C01821=1123.356,380.841,-87.477,-176.868,11.252,149.471
C01822=1123.352,381.088,-87.514,-176.865,11.254,149.471
C01823=1123.349,381.335,-87.552,-176.862,11.256,149.470
C01824=1123.345,381.582,-87.589,-176.859,11.259,149.470
C01825=1123.342,381.830,-87.627,-176.856,11.262,149.470
C01826=1123.338,382.077,-87.664,-176.854,11.263,149.470
C01827=1123.334,382.325,-87.702,-176.851,11.266,149.470
C01828=1123.330,382.571,-87.740,-176.848,11.269,149.470
C01829=1123.326,382.818,-87.777,-176.845,11.272,149.470
C01830=1123.323,383.066,-87.814,-176.842,11.274,149.470
C01831=1123.319,383.313,-87.851,-176.839,11.276,149.470
C01832=1123.315,383.560,-87.889,-176.837,11.278,149.470
C01833=1123.312,383.807,-87.927,-176.835,11.280,149.470
C01834=1123.308,384.054,-87.964,-176.833,11.283,149.470
C01835=1123.304,384.301,-88.002,-176.832,11.284,149.470
C01836=1123.301,384.548,-88.040,-176.830,11.286,149.470
C01837=1123.296,384.796,-88.077,-176.828,11.289,149.470
C01838=1123.293,385.042,-88.115,-176.826,11.291,149.470
C01839=1123.289,385.290,-88.153,-176.824,11.292,149.470
C01840=1123.286,385.536,-88.190,-176.822,11.295,149.470
C01841=1123.282,385.784,-88.227,-176.820,11.297,149.470
C01842=1123.278,386.031,-88.265,-176.819,11.299,149.471
C01843=1123.274,386.278,-88.303,-176.817,11.301,149.471
C01844=1123.271,386.525,-88.341,-176.815,11.303,149.471
C01845=1123.267,386.773,-88.378,-176.814,11.306,149.471
C01846=1123.263,387.019,-88.416,-176.812,11.308,149.471
C01847=1123.260,387.267,-88.454,-176.810,11.310,149.471
C01848=1123.256,387.513,-88.492,-176.809,11.312,149.471
C01849=1123.252,387.761,-88.530,-176.807,11.314,149.471
C01850=1123.248,388.008,-88.567,-176.805,11.317,149.472
C01851=1123.245,388.255,-88.605,-176.803,11.319,149.472
C01852=1123.241,388.502,-88.642,-176.802,11.321,149.472
C01853=1123.238,388.714,-88.675,-176.800,11.323,149.472
C01854=1123.234,388.926,-88.707,-176.799,11.325,149.472
C01855=1123.232,389.138,-88.740,-176.797,11.328,149.473
C01856=1123.228,389.350,-88.773,-176.796,11.329,149.473
C01857=1123.226,389.562,-88.805,-176.795,11.332,149.473
C01858=1123.222,389.775,-88.837,-176.793,11.333,149.473
C01859=1123.219,389.987,-88.870,-176.792,11.336,149.473
C01860=1123.216,390.199,-88.902,-176.791,11.338,149.473
C01861=1123.212,390.446,-88.940,-176.789,11.340,149.474
C01862=1123.209,390.694,-88.978,-176.788,11.343,149.474
C01863=1123.205,390.940,-89.016,-176.786,11.345,149.474
C01864=1123.202,391.188,-89.054,-176.784,11.348,149.475
C01865=1123.197,391.434,-89.092,-176.783,11.351,149.475
C01866=1123.194,391.682,-89.130,-176.781,11.354,149.475
C01867=1123.190,391.928,-89.168,-176.780,11.356,149.475
C01868=1123.187,392.176,-89.206,-176.779,11.358,149.476
C01869=1123.183,392.423,-89.244,-176.778,11.361,149.476
C01870=1123.180,392.670,-89.282,-176.776,11.363,149.476
C01871=1123.176,392.917,-89.320,-176.775,11.366,149.477
C01872=1123.172,393.164,-89.358,-176.773,11.369,149.477
C01873=1123.169,393.411,-89.396,-176.772,11.372,149.477
C01874=1123.164,393.658,-89.434,-176.770,11.374,149.478
C01875=1123.161,393.905,-89.472,-176.769,11.377,149.478
C01876=1123.158,394.153,-89.510,-176.768,11.380,149.479
C01877=1123.153,394.399,-89.548,-176.766,11.383,149.479
C01878=1123.150,394.647,-89.586,-176.765,11.386,149.479
C01879=1123.146,394.893,-89.623,-176.764,11.388,149.480
C01880=1123.142,395.141,-89.662,-176.762,11.392,149.480
C01881=1123.139,395.388,-89.701,-176.761,11.395,149.481
C01882=1123.135,395.634,-89.739,-176.759,11.398,149.481
C01883=1123.132,395.882,-89.777,-176.758,11.401,149.482
C01884=1123.128,396.128,-89.814,-176.757,11.404,149.482
C01885=1123.124,396.376,-89.853,-176.756,11.407,149.482
C01886=1123.121,396.623,-89.891,-176.755,11.410,149.483
C01887=1123.116,396.870,-89.929,-176.753,11.413,149.483
C01888=1123.113,397.117,-89.967,-176.752,11.416,149.484
C01889=1123.110,397.364,-90.005,-176.751,11.419,149.484
C01890=1123.106,397.611,-90.044,-176.750,11.422,149.485
C01891=1123.103,397.858,-90.082,-176.748,11.425,149.485
C01892=1123.099,398.106,-90.120,-176.748,11.429,149.486
C01893=1123.095,398.352,-90.158,-176.747,11.432,149.487
C01894=1123.091,398.599,-90.197,-176.746,11.435,149.487
C01895=1123.088,398.846,-90.235,-176.744,11.439,149.488
C01896=1123.083,399.093,-90.273,-176.743,11.442,149.488
C01897=1123.080,399.341,-90.311,-176.742,11.445,149.489
C01898=1123.077,399.587,-90.350,-176.741,11.448,149.490
C01899=1123.073,399.834,-90.388,-176.740,11.452,149.490
C01900=1123.070,400.081,-90.426,-176.739,11.455,149.491
C01901=1123.066,400.328,-90.465,-176.738,11.459,149.492
C01902=1123.062,400.575,-90.503,-176.737,11.462,149.492
C01903=1123.058,400.823,-90.541,-176.736,11.466,149.493
C01904=1123.055,401.070,-90.579,-176.735,11.469,149.493
C01905=1123.051,401.316,-90.618,-176.734,11.473,149.494
C01906=1123.048,401.563,-90.656,-176.733,11.477,149.495
C01907=1123.044,401.811,-90.694,-176.732,11.480,149.496
C01908=1123.040,402.057,-90.733,-176.732,11.483,149.496
C01909=1123.037,402.270,-90.766,-176.731,11.486,149.497
C01910=1123.034,402.482,-90.799,-176.730,11.490,149.498
C01911=1123.031,402.693,-90.832,-176.729,11.493,149.498
C01912=1123.028,402.906,-90.865,-176.729,11.496,149.499
C01913=1123.024,403.117,-90.898,-176.728,11.500,149.500
C01914=1123.021,403.330,-90.931,-176.727,11.503,149.500
C01915=1123.018,403.541,-90.964,-176.726,11.506,149.501
C01916=1123.015,403.753,-90.997,-176.725,11.509,149.501
C01917=1123.011,404.000,-91.035,-176.725,11.513,149.502
C01918=1123.008,404.247,-91.075,-176.724,11.517,149.503
C01919=1123.005,404.495,-91.112,-176.723,11.521,149.504
C01920=1123.000,404.741,-91.151,-176.722,11.525,149.505
C01921=1122.997,404.988,-91.189,-176.722,11.529,149.506
C01922=1122.993,405.236,-91.228,-176.721,11.533,149.507
C01923=1122.990,405.482,-91.266,-176.720,11.537,149.507
C01924=1122.986,405.729,-91.305,-176.719,11.541,149.508
C01925=1122.982,405.976,-91.344,-176.719,11.545,149.509
C01926=1122.979,406.224,-91.382,-176.719,11.550,149.510
C01927=1122.976,406.470,-91.421,-176.718,11.553,149.511
C01928=1122.972,406.716,-91.459,-176.717,11.558,149.512
C01929=1122.968,406.964,-91.498,-176.716,11.562,149.513
C01930=1122.964,407.211,-91.537,-176.716,11.566,149.514
C01931=1122.961,407.458,-91.575,-176.716,11.571,149.515
C01932=1122.958,407.705,-91.614,-176.715,11.574,149.516
C01933=1122.953,407.952,-91.653,-176.715,11.579,149.517
C01934=1122.950,408.199,-91.691,-176.714,11.584,149.518
C01935=1122.947,408.446,-91.730,-176.714,11.587,149.519
C01936=1122.943,408.693,-91.769,-176.713,11.592,149.520
C01937=1122.940,408.940,-91.808,-176.713,11.597,149.521
C01938=1122.935,409.187,-91.846,-176.712,11.602,149.522
C01939=1122.932,409.434,-91.885,-176.712,11.606,149.523
C01940=1122.929,409.680,-91.924,-176.712,11.611,149.524
C01941=1122.925,409.928,-91.962,-176.711,11.615,149.526
C01942=1122.921,410.175,-92.001,-176.710,11.620,149.527
C01943=1122.918,410.421,-92.040,-176.711,11.624,149.528
C01944=1122.914,410.669,-92.078,-176.710,11.629,149.529
C01945=1122.910,410.915,-92.118,-176.710,11.634,149.530
C01946=1122.907,411.162,-92.157,-176.709,11.639,149.531
C01947=1122.903,411.410,-92.195,-176.709,11.644,149.532
C01948=1122.900,411.657,-92.234,-176.709,11.649,149.534
C01949=1122.896,411.903,-92.273,-176.708,11.654,149.535
C01950=1122.892,412.150,-92.312,-176.709,11.658,149.536
C01951=1122.889,412.397,-92.350,-176.708,11.663,149.537
C01952=1122.885,412.644,-92.389,-176.708,11.668,149.538
C01953=1122.882,412.891,-92.429,-176.708,11.673,149.540
C01954=1122.878,413.138,-92.468,-176.708,11.678,149.541
C01955=1122.875,413.385,-92.506,-176.707,11.683,149.542
C01956=1122.871,413.632,-92.545,-176.707,11.688,149.544
C01957=1122.867,413.879,-92.584,-176.707,11.693,149.545
C01958=1122.865,414.126,-92.623,-176.707,11.699,149.546
C01959=1122.862,414.373,-92.662,-176.707,11.704,149.548
C01960=1122.860,414.620,-92.700,-176.707,11.709,149.549
C01961=1122.859,414.866,-92.739,-176.707,11.714,149.550
C01962=1122.858,415.114,-92.778,-176.707,11.720,149.552
C01963=1122.858,415.361,-92.816,-176.707,11.725,149.553
C01964=1122.858,415.608,-92.855,-176.707,11.730,149.555
C01965=1122.859,415.819,-92.887,-176.707,11.735,149.556
C01966=1122.860,416.031,-92.920,-176.708,11.740,149.557
C01967=1122.862,416.243,-92.953,-176.707,11.745,149.558
C01968=1122.864,416.455,-92.986,-176.708,11.749,149.560
C01969=1122.865,416.667,-93.019,-176.708,11.754,149.561
C01970=1122.869,416.878,-93.052,-176.708,11.759,149.562
C01971=1122.872,417.090,-93.084,-176.708,11.764,149.564
C01972=1122.876,417.302,-93.116,-176.709,11.768,149.565
C01973=1122.457,417.301,-93.179,-176.701,11.773,149.564
C01974=1122.453,417.090,-93.147,-176.701,11.768,149.563
C01975=1122.449,416.878,-93.114,-176.701,11.763,149.561
C01976=1122.447,416.667,-93.081,-176.700,11.759,149.560
C01977=1122.445,416.455,-93.049,-176.700,11.753,149.559
C01978=1122.443,416.243,-93.016,-176.700,11.749,149.558
C01979=1122.441,416.031,-92.983,-176.700,11.744,149.556
C01980=1122.440,415.819,-92.950,-176.700,11.740,149.555
C01981=1122.439,415.607,-92.917,-176.700,11.735,149.554
C01982=1122.438,415.360,-92.879,-176.700,11.730,149.553
C01983=1122.439,415.113,-92.840,-176.700,11.724,149.551
C01984=1122.440,414.867,-92.801,-176.700,11.719,149.550
C01985=1122.441,414.620,-92.763,-176.700,11.714,149.548
C01986=1122.443,414.373,-92.724,-176.700,11.709,149.547
C01987=1122.445,414.125,-92.685,-176.700,11.703,149.546
C01988=1122.448,413.879,-92.647,-176.701,11.697,149.544
C01989=1122.452,413.632,-92.607,-176.701,11.692,149.543
C01990=1122.455,413.385,-92.568,-176.701,11.687,149.542
C01991=1122.458,413.138,-92.529,-176.701,11.682,149.540
C01992=1122.462,412.891,-92.490,-176.701,11.677,149.539
C01993=1122.466,412.643,-92.452,-176.702,11.672,149.538
C01994=1122.470,412.397,-92.413,-176.702,11.667,149.537
C01995=1122.473,412.150,-92.374,-176.702,11.662,149.536
C01996=1122.476,411.904,-92.335,-176.703,11.657,149.534
C01997=1122.480,411.656,-92.296,-176.703,11.652,149.533
C01998=1122.484,411.409,-92.257,-176.703,11.647,149.532
C01999=1122.488,411.162,-92.218,-176.703,11.643,149.531
C02000=1122.490,410.915,-92.179,-176.703,11.638,149.529
C02001=1122.495,410.668,-92.141,-176.704,11.633,149.528
C02002=1122.499,410.422,-92.102,-176.704,11.628,149.527
C02003=1122.501,410.175,-92.063,-176.705,11.623,149.526
C02004=1122.505,409.927,-92.025,-176.705,11.618,149.525
C02005=1122.509,409.680,-91.985,-176.706,11.614,149.524
C02006=1122.513,409.433,-91.946,-176.706,11.610,149.523
C02007=1122.516,409.187,-91.909,-176.706,11.605,149.522
C02008=1122.520,408.940,-91.869,-176.707,11.600,149.521
C02009=1122.524,408.693,-91.830,-176.708,11.596,149.520
C02010=1122.527,408.446,-91.792,-176.708,11.591,149.518
C02011=1122.530,408.199,-91.753,-176.708,11.587,149.517
C02012=1122.535,407.952,-91.714,-176.709,11.582,149.517
C02013=1122.538,407.705,-91.676,-176.710,11.578,149.515
C02014=1122.541,407.458,-91.637,-176.710,11.574,149.515
C02015=1122.545,407.211,-91.598,-176.711,11.570,149.514
C02016=1122.548,406.964,-91.560,-176.712,11.565,149.512
C02017=1122.552,406.718,-91.521,-176.713,11.560,149.512
C02018=1122.556,406.470,-91.482,-176.713,11.557,149.511
C02019=1122.559,406.223,-91.444,-176.714,11.552,149.510
C02020=1122.563,405.976,-91.405,-176.714,11.549,149.509
C02021=1122.567,405.730,-91.367,-176.715,11.544,149.508
C02022=1122.571,405.482,-91.328,-176.716,11.540,149.507
C02023=1122.574,405.235,-91.289,-176.716,11.536,149.506
C02024=1122.577,404.988,-91.251,-176.717,11.532,149.505
C02025=1122.581,404.741,-91.212,-176.718,11.528,149.504
C02026=1122.585,404.495,-91.174,-176.719,11.524,149.504
C02027=1122.588,404.248,-91.135,-176.719,11.520,149.503
C02028=1122.592,404.000,-91.096,-176.720,11.516,149.502
C02029=1122.595,403.753,-91.058,-176.721,11.512,149.501
C02030=1122.599,403.541,-91.025,-176.722,11.509,149.500
C02031=1122.602,403.329,-90.992,-176.722,11.506,149.500
C02032=1122.605,403.118,-90.958,-176.723,11.502,149.499
C02033=1122.609,402.905,-90.926,-176.724,11.499,149.498
C02034=1122.611,402.694,-90.893,-176.725,11.496,149.498
C02035=1122.614,402.482,-90.861,-176.726,11.493,149.497
C02036=1122.618,402.270,-90.827,-176.726,11.489,149.496
C02037=1122.621,402.058,-90.794,-176.727,11.486,149.496
C02038=1122.625,401.810,-90.755,-176.729,11.482,149.495
C02039=1122.628,401.563,-90.718,-176.729,11.479,149.495
C02040=1122.632,401.316,-90.678,-176.730,11.475,149.494
C02041=1122.635,401.070,-90.641,-176.731,11.471,149.493
C02042=1122.639,400.823,-90.601,-176.732,11.468,149.492
C02043=1122.642,400.575,-90.564,-176.733,11.464,149.492
C02044=1122.647,400.329,-90.525,-176.735,11.461,149.491
C02045=1122.650,400.081,-90.487,-176.735,11.458,149.490
C02046=1122.653,399.834,-90.448,-176.736,11.454,149.490
C02047=1122.657,399.588,-90.411,-176.738,11.450,149.489
C02048=1122.661,399.340,-90.372,-176.738,11.447,149.489
C02049=1122.664,399.094,-90.333,-176.739,11.444,149.488
C02050=1122.669,398.847,-90.295,-176.741,11.440,149.487
C02051=1122.672,398.599,-90.257,-176.742,11.437,149.487
C02052=1122.675,398.352,-90.219,-176.743,11.434,149.486
C02053=1122.679,398.106,-90.180,-176.744,11.431,149.486
C02054=1122.682,397.859,-90.143,-176.746,11.427,149.485
C02055=1122.686,397.611,-90.104,-176.747,11.424,149.485
C02056=1122.690,397.364,-90.066,-176.748,11.421,149.484
C02057=1122.694,397.117,-90.028,-176.749,11.418,149.484
C02058=1122.697,396.870,-89.989,-176.750,11.415,149.483
C02059=1122.701,396.623,-89.951,-176.752,11.411,149.483
C02060=1122.705,396.376,-89.913,-176.753,11.408,149.482
C02061=1122.708,396.129,-89.876,-176.754,11.405,149.482
C02062=1122.712,395.882,-89.837,-176.756,11.403,149.481
C02063=1122.715,395.635,-89.799,-176.757,11.400,149.481
C02064=1122.720,395.388,-89.761,-176.758,11.397,149.480
C02065=1122.723,395.141,-89.722,-176.759,11.394,149.480
C02066=1122.726,394.894,-89.684,-176.761,11.390,149.479
C02067=1122.731,394.647,-89.646,-176.762,11.387,149.479
C02068=1122.734,394.400,-89.608,-176.763,11.384,149.479
C02069=1122.738,394.153,-89.571,-176.765,11.382,149.478
C02070=1122.742,393.906,-89.532,-176.766,11.379,149.478
C02071=1122.745,393.658,-89.494,-176.768,11.376,149.477
C02072=1122.749,393.411,-89.456,-176.769,11.373,149.477
C02073=1122.752,393.164,-89.418,-176.771,11.371,149.477
C02074=1122.756,392.918,-89.380,-176.772,11.368,149.476
C02075=1122.760,392.670,-89.342,-176.773,11.365,149.476
C02076=1122.764,392.423,-89.304,-176.775,11.363,149.476
C02077=1122.767,392.176,-89.266,-176.776,11.360,149.476
C02078=1122.771,391.929,-89.228,-176.778,11.357,149.475
C02079=1122.775,391.682,-89.190,-176.779,11.354,149.475
C02080=1122.778,391.435,-89.152,-176.781,11.352,149.475
C02081=1122.782,391.188,-89.115,-176.782,11.349,149.474
C02082=1122.786,390.941,-89.076,-176.784,11.347,149.474
C02083=1122.790,390.694,-89.039,-176.786,11.344,149.474
C02084=1122.793,390.447,-89.001,-176.787,11.341,149.473
C02085=1122.796,390.199,-88.963,-176.789,11.339,149.473
C02086=1122.799,389.987,-88.930,-176.790,11.337,149.473
C02087=1122.803,389.775,-88.898,-176.792,11.335,149.473
C02088=1122.806,389.563,-88.866,-176.793,11.333,149.473
C02089=1122.809,389.351,-88.832,-176.795,11.330,149.473
C02090=1122.812,389.139,-88.800,-176.796,11.329,149.472
C02091=1122.815,388.927,-88.768,-176.797,11.326,149.472
C02092=1122.819,388.715,-88.736,-176.799,11.325,149.472
C02093=1122.822,388.503,-88.704,-176.800,11.322,149.472
C02094=1122.826,388.255,-88.665,-176.801,11.320,149.472
C02095=1122.829,388.008,-88.627,-176.803,11.318,149.471
C02096=1122.833,387.762,-88.590,-176.805,11.316,149.471
C02097=1122.836,387.514,-88.552,-176.807,11.313,149.471
C02098=1122.840,387.267,-88.515,-176.809,11.311,149.471
C02099=1122.844,387.019,-88.476,-176.811,11.309,149.471
C02100=1122.848,386.773,-88.439,-176.812,11.307,149.471
C02101=1122.851,386.526,-88.401,-176.814,11.305,149.471
C02102=1122.855,386.278,-88.364,-176.816,11.302,149.471
C02103=1122.858,386.031,-88.326,-176.817,11.300,149.470
C02104=1122.863,385.784,-88.288,-176.819,11.298,149.470
C02105=1122.866,385.537,-88.250,-176.821,11.296,149.470
C02106=1122.870,385.290,-88.213,-176.822,11.294,149.470
C02107=1122.874,385.043,-88.175,-176.825,11.292,149.470
C02108=1122.877,384.796,-88.137,-176.827,11.289,149.470
C02109=1122.881,384.549,-88.100,-176.829,11.287,149.470
C02110=1122.884,384.302,-88.063,-176.830,11.286,149.470
C02111=1122.889,384.055,-88.024,-176.832,11.283,149.470
C02112=1122.892,383.807,-87.986,-176.834,11.281,149.470
C02113=1122.896,383.560,-87.950,-176.836,11.279,149.470
C02114=1122.899,383.313,-87.912,-176.838,11.277,149.470
C02115=1122.903,383.066,-87.874,-176.841,11.275,149.470
C02116=1122.906,382.818,-87.837,-176.844,11.272,149.470
C02117=1122.910,382.572,-87.799,-176.847,11.270,149.470
C02118=1122.914,382.325,-87.762,-176.850,11.267,149.470
C02119=1122.918,382.077,-87.725,-176.852,11.265,149.470
C02120=1122.921,381.831,-87.687,-176.855,11.262,149.470
C02121=1122.926,381.583,-87.649,-176.858,11.259,149.470
C02122=1122.929,381.336,-87.612,-176.862,11.257,149.471
C02123=1122.933,381.088,-87.574,-176.864,11.255,149.471
C02124=1122.937,380.842,-87.537,-176.867,11.252,149.471
C02125=1122.941,380.594,-87.500,-176.870,11.250,149.471
C02126=1122.944,380.347,-87.462,-176.873,11.247,149.471
C02127=1122.948,380.100,-87.425,-176.876,11.244,149.471
C02128=1122.952,379.853,-87.388,-176.879,11.243,149.471
C02129=1122.955,379.606,-87.350,-176.882,11.240,149.471
C02130=1122.959,379.359,-87.313,-176.885,11.237,149.471
C02131=1122.963,379.111,-87.275,-176.888,11.234,149.471
C02132=1122.966,378.865,-87.238,-176.891,11.233,149.472
C02133=1122.970,378.617,-87.201,-176.894,11.230,149.472
C02134=1122.974,378.369,-87.164,-176.897,11.227,149.472
C02135=1122.978,378.123,-87.126,-176.900,11.225,149.472
C02136=1122.982,377.876,-87.089,-176.902,11.223,149.472
C02137=1122.985,377.628,-87.053,-176.906,11.220,149.472
C02138=1122.988,377.382,-87.015,-176.909,11.218,149.473
C02139=1122.992,377.134,-86.978,-176.912,11.215,149.473
C02140=1122.996,376.886,-86.941,-176.915,11.213,149.473
C02141=1123.000,376.640,-86.904,-176.918,11.211,149.473
C02142=1123.004,376.427,-86.872,-176.921,11.208,149.473
C02143=1123.007,376.216,-86.840,-176.923,11.206,149.473
C02144=1123.010,376.003,-86.809,-176.926,11.204,149.473
C02145=1123.013,375.791,-86.776,-176.928,11.203,149.474
C02146=1123.016,375.579,-86.744,-176.931,11.200,149.474
C02147=1123.019,375.366,-86.713,-176.934,11.198,149.474
C02148=1123.023,375.155,-86.681,-176.936,11.196,149.474
C02149=1123.026,374.942,-86.649,-176.939,11.195,149.474
C02150=1123.030,374.694,-86.612,-176.942,11.192,149.474
C02151=1123.033,374.447,-86.575,-176.945,11.190,149.475
C02152=1123.037,374.200,-86.538,-176.948,11.187,149.475
C02153=1123.041,373.953,-86.502,-176.952,11.184,149.475
C02154=1123.045,373.705,-86.464,-176.954,11.183,149.475
C02155=1123.049,373.458,-86.427,-176.958,11.180,149.475
C02156=1123.052,373.211,-86.391,-176.961,11.178,149.475
C02157=1123.056,372.964,-86.354,-176.964,11.175,149.476
C02158=1123.060,372.716,-86.317,-176.968,11.173,149.476
C02159=1123.064,372.469,-86.280,-176.970,11.171,149.476
C02160=1123.067,372.222,-86.244,-176.974,11.169,149.476
C02161=1123.071,371.975,-86.206,-176.977,11.166,149.477
C02162=1123.075,371.728,-86.170,-176.980,11.163,149.477
C02163=1123.078,371.480,-86.132,-176.983,11.161,149.477
C02164=1123.082,371.233,-86.097,-176.986,11.158,149.477
C02165=1123.086,370.986,-86.060,-176.989,11.157,149.477
C02166=1123.090,370.738,-86.023,-176.992,11.154,149.477
C02167=1123.094,370.492,-85.987,-176.996,11.152,149.478
C02168=1123.097,370.244,-85.950,-176.999,11.149,149.478
C02169=1123.101,369.996,-85.913,-177.002,11.147,149.478
C02170=1123.105,369.750,-85.876,-177.005,11.144,149.478
C02171=1123.109,369.502,-85.840,-177.009,11.143,149.479
C02172=1123.113,369.255,-85.803,-177.012,11.140,149.479
C02173=1123.116,369.008,-85.766,-177.015,11.138,149.479
C02174=1123.120,368.760,-85.729,-177.018,11.135,149.479
C02175=1123.124,368.513,-85.693,-177.022,11.133,149.479
C02176=1123.127,368.266,-85.657,-177.025,11.130,149.480
C02177=1123.131,368.019,-85.620,-177.028,11.128,149.480
C02178=1123.135,367.772,-85.584,-177.032,11.125,149.480
C02179=1123.139,367.524,-85.548,-177.034,11.124,149.480
C02180=1123.143,367.277,-85.511,-177.038,11.121,149.481
C02181=1123.147,367.030,-85.474,-177.041,11.119,149.481
C02182=1123.150,366.782,-85.437,-177.044,11.116,149.481
C02183=1123.154,366.534,-85.402,-177.048,11.114,149.481
C02184=1123.158,366.287,-85.365,-177.051,11.112,149.482
C02185=1123.161,366.040,-85.329,-177.055,11.109,149.482
C02186=1123.166,365.793,-85.292,-177.058,11.107,149.482
C02187=1123.169,365.546,-85.256,-177.061,11.104,149.482
C02188=1123.173,365.298,-85.219,-177.064,11.103,149.483
C02189=1123.177,365.051,-85.184,-177.067,11.100,149.483
C02190=1123.181,364.804,-85.147,-177.071,11.098,149.483
C02191=1123.185,364.556,-85.111,-177.074,11.096,149.483
C02192=1123.189,364.309,-85.074,-177.077,11.093,149.484
C02193=1123.192,364.062,-85.038,-177.081,11.091,149.484
C02194=1123.196,363.814,-85.002,-177.084,11.088,149.484
C02195=1123.199,363.567,-84.965,-177.088,11.086,149.484
C02196=1123.204,363.319,-84.929,-177.091,11.084,149.485
C02197=1123.207,363.072,-84.893,-177.094,11.081,149.485
C02198=1123.211,362.826,-84.857,-177.098,11.079,149.485
C02199=1123.215,362.580,-84.821,-177.101,11.076,149.485
C02200=1123.218,362.332,-84.786,-177.105,11.074,149.486
C02201=1123.222,362.086,-84.750,-177.108,11.071,149.486
C02202=1123.226,361.839,-84.714,-177.111,11.069,149.486
C02203=1123.230,361.593,-84.678,-177.115,11.067,149.486
C02204=1123.234,361.347,-84.642,-177.118,11.064,149.486
C02205=1123.237,361.100,-84.605,-177.122,11.062,149.487
C02206=1123.241,360.852,-84.569,-177.125,11.059,149.487
C02207=1123.245,360.605,-84.534,-177.128,11.057,149.487
C02208=1123.248,360.358,-84.498,-177.131,11.055,149.488
C02209=1123.253,360.110,-84.461,-177.135,11.052,149.488
C02210=1123.257,359.863,-84.426,-177.138,11.050,149.488
C02211=1123.260,359.616,-84.390,-177.142,11.047,149.488
C02212=1123.264,359.368,-84.354,-177.145,11.045,149.489
C02213=1123.268,359.120,-84.318,-177.148,11.043,149.489
C02214=1123.272,358.874,-84.283,-177.152,11.040,149.489
C02215=1123.276,358.627,-84.246,-177.155,11.038,149.489
C02216=1123.279,358.379,-84.211,-177.159,11.035,149.490
C02217=1123.284,358.131,-84.175,-177.162,11.033,149.490
C02218=1123.287,357.884,-84.139,-177.166,11.031,149.490
C02219=1123.291,357.636,-84.104,-177.169,11.028,149.490
C02220=1123.294,357.389,-84.067,-177.172,11.026,149.491
C02221=1123.299,357.142,-84.031,-177.176,11.023,149.491
C02222=1123.302,356.928,-84.001,-177.179,11.021,149.491
C02223=1123.305,356.715,-83.970,-177.182,11.019,149.491
C02224=1123.309,356.502,-83.940,-177.185,11.017,149.492
C02225=1123.312,356.289,-83.909,-177.188,11.015,149.492
C02226=1123.315,356.076,-83.878,-177.191,11.013,149.492
C02227=1123.319,355.863,-83.847,-177.194,11.010,149.492
C02228=1123.322,355.649,-83.817,-177.197,11.009,149.493
C02229=1123.325,355.435,-83.786,-177.200,11.006,149.493
C02230=1123.329,355.189,-83.750,-177.204,11.004,149.493
C02231=1123.333,354.941,-83.715,-177.207,11.001,149.493
C02232=1123.336,354.694,-83.679,-177.210,10.999,149.493
C02233=1123.341,354.446,-83.643,-177.214,10.997,149.494
C02234=1123.344,354.198,-83.608,-177.217,10.994,149.494
C02235=1123.348,353.951,-83.572,-177.221,10.991,149.494
C02236=1123.352,353.704,-83.537,-177.224,10.988,149.495
C02237=1123.356,353.456,-83.501,-177.228,10.986,149.495
C02238=1123.360,353.209,-83.466,-177.231,10.984,149.495
C02239=1123.363,352.961,-83.430,-177.235,10.981,149.495
C02240=1123.367,352.713,-83.395,-177.238,10.979,149.496
C02241=1123.371,352.467,-83.360,-177.242,10.976,149.496
C02242=1123.375,352.219,-83.325,-177.246,10.973,149.496
C02243=1123.379,351.972,-83.289,-177.249,10.971,149.496
C02244=1123.382,351.724,-83.254,-177.252,10.969,149.497
C02245=1123.387,351.477,-83.219,-177.256,10.965,149.497
C02246=1123.391,351.229,-83.184,-177.260,10.963,149.497
C02247=1123.394,350.982,-83.148,-177.263,10.960,149.497
C02248=1123.398,350.734,-83.113,-177.267,10.958,149.498
C02249=1123.403,350.487,-83.078,-177.271,10.955,149.498
C02250=1123.406,350.239,-83.043,-177.274,10.953,149.498
C02251=1123.410,349.992,-83.007,-177.277,10.950,149.498
C02252=1123.414,349.745,-82.972,-177.280,10.948,149.499
C02253=1123.418,349.497,-82.937,-177.284,10.944,149.499
C02254=1123.421,349.284,-82.907,-177.287,10.943,149.499
C02255=1123.424,349.072,-82.876,-177.289,10.941,149.499
C02256=1123.428,348.860,-82.847,-177.293,10.938,149.499
C02257=1123.431,348.646,-82.816,-177.295,10.937,149.500
C02258=1123.434,348.434,-82.786,-177.298,10.934,149.500
C02259=1123.438,348.221,-82.756,-177.301,10.932,149.500
C02260=1123.441,348.009,-82.726,-177.304,10.930,149.500
C02261=1123.445,347.796,-82.696,-177.307,10.928,149.500
C02262=1123.448,347.548,-82.660,-177.310,10.925,149.500
C02263=1123.453,347.301,-82.626,-177.313,10.923,149.501
C02264=1123.457,347.054,-82.590,-177.317,10.920,149.501
C02265=1123.460,346.806,-82.556,-177.320,10.918,149.501
C02266=1123.464,346.559,-82.521,-177.323,10.915,149.501
C02267=1123.468,346.311,-82.486,-177.325,10.913,149.501
C02268=1123.472,346.064,-82.451,-177.329,10.911,149.502
C02269=1123.476,345.816,-82.416,-177.332,10.908,149.502
C02270=1123.479,345.569,-82.381,-177.335,10.906,149.502
C02271=1123.484,345.321,-82.347,-177.339,10.903,149.502
C02272=1123.487,345.074,-82.311,-177.342,10.901,149.502
C02273=1123.492,344.826,-82.277,-177.345,10.898,149.503
C02274=1123.496,344.578,-82.242,-177.348,10.896,149.503
C02275=1123.499,344.331,-82.207,-177.352,10.893,149.503
C02276=1123.503,344.084,-82.172,-177.355,10.891,149.503
C02277=1123.507,343.836,-82.138,-177.358,10.888,149.504
C02278=1123.512,343.589,-82.102,-177.361,10.886,149.504
C02279=1123.515,343.341,-82.068,-177.364,10.883,149.504
C02280=1123.519,343.093,-82.033,-177.368,10.881,149.504
C02281=1123.523,342.845,-81.999,-177.371,10.878,149.504
C02282=1123.526,342.598,-81.964,-177.374,10.876,149.505
C02283=1123.531,342.351,-81.930,-177.378,10.873,149.505
C02284=1123.535,342.103,-81.895,-177.380,10.871,149.505
C02285=1123.539,341.856,-81.861,-177.383,10.869,149.505
C02286=1123.542,341.608,-81.825,-177.387,10.866,149.505
C02287=1123.547,341.361,-81.791,-177.390,10.864,149.506
C02288=1123.550,341.113,-81.757,-177.393,10.862,149.506
C02289=1123.555,340.865,-81.722,-177.396,10.859,149.506
C02290=1123.559,340.617,-81.687,-177.399,10.856,149.506
C02291=1123.563,340.370,-81.653,-177.403,10.854,149.506
C02292=1123.567,340.122,-81.619,-177.406,10.851,149.507
C02293=1123.570,339.876,-81.584,-177.409,10.849,149.507
C02294=1123.574,339.627,-81.549,-177.412,10.846,149.507
C02295=1123.579,339.380,-81.515,-177.416,10.844,149.507
C02296=1123.582,339.132,-81.480,-177.419,10.841,149.507
C02297=1123.586,338.885,-81.446,-177.422,10.839,149.508
C02298=1123.590,338.637,-81.412,-177.426,10.836,149.508
C02299=1123.594,338.390,-81.377,-177.428,10.834,149.508
C02300=1123.597,338.142,-81.343,-177.432,10.831,149.508
C02301=1123.602,337.894,-81.309,-177.435,10.829,149.508
C02302=1123.606,337.647,-81.275,-177.438,10.827,149.509
C02303=1123.610,337.399,-81.240,-177.441,10.824,149.509
C02304=1123.614,337.152,-81.206,-177.444,10.822,149.509
C02305=1123.618,336.904,-81.171,-177.447,10.819,149.509
C02306=1123.622,336.656,-81.138,-177.451,10.817,149.509
C02307=1123.626,336.408,-81.103,-177.454,10.814,149.509
C02308=1123.630,336.161,-81.069,-177.457,10.812,149.510
C02309=1123.634,335.913,-81.035,-177.460,10.809,149.510
C02310=1123.637,335.701,-81.005,-177.463,10.807,149.510
C02311=1123.640,335.488,-80.976,-177.466,10.805,149.510
C02312=1123.643,335.275,-80.946,-177.469,10.803,149.510
C02313=1123.647,335.062,-80.917,-177.471,10.800,149.510
C02314=1123.650,334.850,-80.888,-177.474,10.799,149.511
C02315=1123.654,334.637,-80.859,-177.476,10.797,149.511
C02316=1123.657,334.424,-80.830,-177.480,10.794,149.511
C02317=1123.660,334.212,-80.801,-177.482,10.792,149.511
C02318=1123.664,333.964,-80.766,-177.485,10.790,149.511
C02319=1123.669,333.716,-80.733,-177.489,10.787,149.512
C02320=1123.673,333.469,-80.698,-177.492,10.784,149.512
C02321=1123.676,333.221,-80.664,-177.495,10.782,149.512
C02322=1123.681,332.973,-80.631,-177.498,10.779,149.512
C02323=1123.684,332.725,-80.596,-177.501,10.777,149.512
C02324=1123.688,332.478,-80.562,-177.504,10.774,149.512
C02325=1123.692,332.230,-80.529,-177.508,10.772,149.513
C02326=1123.696,331.983,-80.495,-177.511,10.769,149.513
C02327=1123.700,331.735,-80.460,-177.514,10.767,149.513
C02328=1123.704,331.487,-80.427,-177.517,10.765,149.513
C02329=1123.708,331.240,-80.393,-177.520,10.762,149.514
C02330=1123.712,330.992,-80.359,-177.523,10.760,149.514
C02331=1123.716,330.745,-80.325,-177.526,10.757,149.514
C02332=1123.720,330.497,-80.291,-177.530,10.755,149.514
C02333=1123.724,330.249,-80.258,-177.533,10.752,149.514
C02334=1123.728,330.002,-80.223,-177.536,10.750,149.514
C02335=1123.732,329.754,-80.190,-177.539,10.747,149.515
C02336=1123.736,329.506,-80.156,-177.542,10.745,149.515
C02337=1123.740,329.258,-80.123,-177.546,10.742,149.515
C02338=1123.744,329.011,-80.089,-177.549,10.739,149.515
C02339=1123.748,328.763,-80.055,-177.552,10.737,149.515
C02340=1123.752,328.515,-80.021,-177.555,10.735,149.516
C02341=1123.756,328.268,-79.988,-177.558,10.732,149.516
C02342=1123.760,328.020,-79.955,-177.562,10.729,149.516
C02343=1123.764,327.773,-79.921,-177.565,10.727,149.516
C02344=1123.768,327.525,-79.887,-177.567,10.725,149.516
C02345=1123.772,327.276,-79.853,-177.571,10.722,149.517
C02346=1123.776,327.029,-79.819,-177.574,10.720,149.517
C02347=1123.780,326.781,-79.786,-177.577,10.718,149.517
C02348=1123.784,326.534,-79.752,-177.580,10.715,149.517
C02349=1123.788,326.286,-79.719,-177.583,10.712,149.517
C02350=1123.792,326.038,-79.686,-177.587,10.710,149.518
C02351=1123.796,325.790,-79.653,-177.590,10.707,149.518
C02352=1123.800,325.543,-79.619,-177.593,10.705,149.518
C02353=1123.804,325.296,-79.586,-177.596,10.702,149.518
C02354=1123.807,325.047,-79.552,-177.599,10.699,149.518
C02355=1123.811,324.799,-79.519,-177.603,10.697,149.518
C02356=1123.816,324.552,-79.484,-177.606,10.695,149.519
C02357=1123.820,324.304,-79.451,-177.609,10.692,149.519
C02358=1123.824,324.057,-79.418,-177.612,10.689,149.519
C02359=1123.828,323.809,-79.385,-177.615,10.687,149.519
C02360=1123.833,323.561,-79.352,-177.618,10.685,149.519
C02361=1123.836,323.313,-79.318,-177.621,10.682,149.520
C02362=1123.839,323.066,-79.285,-177.624,10.680,149.520
C02363=1123.843,322.818,-79.252,-177.627,10.677,149.520
C02364=1123.848,322.570,-79.219,-177.631,10.675,149.520
C02365=1123.852,322.323,-79.186,-177.634,10.672,149.520
C02366=1123.855,322.110,-79.157,-177.636,10.670,149.521
C02367=1123.859,321.896,-79.129,-177.639,10.668,149.521
C02368=1123.862,321.684,-79.100,-177.642,10.666,149.521
C02369=1123.865,321.471,-79.071,-177.645,10.663,149.521
C02370=1123.869,321.258,-79.042,-177.648,10.661,149.521
C02371=1123.872,321.045,-79.014,-177.650,10.659,149.521
C02372=1123.876,320.833,-78.986,-177.653,10.657,149.522
C02373=1123.880,320.620,-78.957,-177.655,10.655,149.522
C02374=1123.884,320.372,-78.924,-177.659,10.653,149.522
C02375=1123.888,320.124,-78.891,-177.662,10.650,149.522
C02376=1123.891,319.876,-78.858,-177.665,10.647,149.522
C02377=1123.895,319.628,-78.825,-177.668,10.645,149.522
C02378=1123.899,319.381,-78.792,-177.671,10.642,149.523
C02379=1123.903,319.133,-78.759,-177.675,10.640,149.523
C02380=1123.907,318.885,-78.726,-177.678,10.637,149.523
C02381=1123.912,318.637,-78.693,-177.681,10.634,149.523
C02382=1123.915,318.389,-78.661,-177.684,10.632,149.523
C02383=1123.919,318.142,-78.627,-177.686,10.630,149.523
C02384=1123.923,317.894,-78.594,-177.690,10.628,149.524
C02385=1123.927,317.646,-78.561,-177.693,10.625,149.524
C02386=1123.932,317.399,-78.528,-177.696,10.622,149.524
C02387=1123.935,317.151,-78.496,-177.699,10.620,149.524
C02388=1123.939,316.903,-78.463,-177.702,10.617,149.524
C02389=1123.944,316.655,-78.430,-177.706,10.615,149.525
C02390=1123.948,316.407,-78.397,-177.709,10.612,149.525
C02391=1123.951,316.159,-78.365,-177.712,10.609,149.525
C02392=1123.956,315.912,-78.332,-177.715,10.607,149.525
C02393=1123.960,315.664,-78.299,-177.718,10.604,149.525
C02394=1123.963,315.416,-78.267,-177.721,10.602,149.525
C02395=1123.968,315.168,-78.234,-177.725,10.599,149.526
C02396=1123.972,314.920,-78.200,-177.728,10.597,149.526
C02397=1123.975,314.672,-78.169,-177.730,10.595,149.526
C02398=1123.980,314.425,-78.135,-177.733,10.592,149.526
C02399=1123.984,314.177,-78.102,-177.737,10.590,149.526
C02400=1123.987,313.929,-78.070,-177.740,10.587,149.527
C02401=1123.991,313.681,-78.037,-177.743,10.585,149.527
C02402=1123.996,313.433,-78.005,-177.746,10.582,149.527
C02403=1124.000,313.186,-77.973,-177.749,10.579,149.527
C02404=1124.004,312.938,-77.939,-177.752,10.577,149.527
C02405=1124.009,312.690,-77.907,-177.756,10.574,149.528
C02406=1124.012,312.443,-77.874,-177.759,10.572,149.528
C02407=1124.016,312.194,-77.842,-177.762,10.569,149.528
C02408=1124.020,311.947,-77.809,-177.765,10.566,149.528
C02409=1124.024,311.698,-77.777,-177.768,10.564,149.528
C02410=1124.028,311.451,-77.744,-177.771,10.561,149.528
C02411=1124.032,311.203,-77.712,-177.774,10.560,149.529
C02412=1124.037,310.955,-77.680,-177.777,10.557,149.529
C02413=1124.040,310.708,-77.647,-177.780,10.554,149.529
C02414=1124.045,310.459,-77.615,-177.784,10.552,149.529
C02415=1124.048,310.212,-77.582,-177.786,10.549,149.529
C02416=1124.053,309.963,-77.550,-177.790,10.547,149.530
C02417=1124.056,309.715,-77.518,-177.793,10.544,149.530
C02418=1124.061,309.468,-77.485,-177.796,10.542,149.530
C02419=1124.065,309.220,-77.453,-177.799,10.539,149.530
C02420=1124.069,308.972,-77.421,-177.802,10.536,149.530
C02421=1124.073,308.725,-77.388,-177.806,10.534,149.530
C02422=1124.077,308.511,-77.360,-177.808,10.532,149.531
C02423=1124.080,308.299,-77.333,-177.810,10.530,149.531
C02424=1124.083,308.085,-77.305,-177.814,10.527,149.531
C02425=1124.087,307.872,-77.277,-177.816,10.525,149.531
C02426=1124.091,307.659,-77.250,-177.819,10.523,149.531
C02427=1124.094,307.446,-77.223,-177.822,10.521,149.531
C02428=1124.098,307.233,-77.194,-177.824,10.519,149.532
C02429=1124.102,307.020,-77.167,-177.827,10.516,149.532
C02430=1124.105,306.772,-77.135,-177.830,10.514,149.532
C02431=1124.109,306.524,-77.102,-177.833,10.511,149.532
C02432=1124.113,306.276,-77.070,-177.836,10.509,149.532
C02433=1124.117,306.029,-77.039,-177.839,10.507,149.532
C02434=1124.122,305.781,-77.006,-177.842,10.504,149.533
C02435=1124.126,305.533,-76.975,-177.845,10.502,149.533
C02436=1124.130,305.284,-76.942,-177.848,10.499,149.533
C02437=1124.134,305.037,-76.911,-177.852,10.497,149.533
C02438=1124.138,304.789,-76.879,-177.854,10.494,149.533
C02439=1124.142,304.541,-76.846,-177.858,10.491,149.534
C02440=1124.146,304.294,-76.814,-177.861,10.489,149.534
C02441=1124.150,304.046,-76.782,-177.864,10.486,149.534
C02442=1124.155,303.798,-76.750,-177.867,10.483,149.534
C02443=1124.158,303.549,-76.718,-177.870,10.481,149.534
C02444=1124.163,303.302,-76.687,-177.873,10.479,149.534
C02445=1124.166,303.054,-76.655,-177.876,10.477,149.535
C02446=1124.171,302.806,-76.622,-177.879,10.474,149.535
C02447=1124.175,302.558,-76.591,-177.882,10.471,149.535
C02448=1124.179,302.310,-76.560,-177.886,10.469,149.535
C02449=1124.184,302.061,-76.527,-177.889,10.466,149.535
C02450=1124.188,301.814,-76.496,-177.892,10.464,149.536
C02451=1124.192,301.566,-76.464,-177.895,10.461,149.536
C02452=1124.195,301.318,-76.432,-177.898,10.459,149.536
C02453=1124.200,301.071,-76.401,-177.901,10.456,149.536
C02454=1124.204,300.822,-76.368,-177.904,10.453,149.536
C02455=1124.208,300.574,-76.336,-177.907,10.451,149.536
C02456=1124.212,300.326,-76.305,-177.911,10.448,149.537
C02457=1124.216,300.078,-76.274,-177.913,10.446,149.537
C02458=1124.220,299.831,-76.242,-177.916,10.444,149.537
C02459=1124.225,299.583,-76.210,-177.919,10.441,149.537
C02460=1124.228,299.335,-76.178,-177.923,10.439,149.537
C02461=1124.233,299.087,-76.147,-177.925,10.436,149.537
C02462=1124.237,298.839,-76.115,-177.929,10.433,149.538
C02463=1124.240,298.590,-76.083,-177.932,10.431,149.538
C02464=1124.245,298.343,-76.052,-177.935,10.428,149.538
C02465=1124.249,298.095,-76.021,-177.938,10.425,149.538
C02466=1124.253,297.847,-75.989,-177.941,10.423,149.538
C02467=1124.257,297.599,-75.957,-177.944,10.420,149.538
C02468=1124.262,297.351,-75.926,-177.947,10.419,149.539
C02469=1124.266,297.103,-75.894,-177.950,10.416,149.539
C02470=1124.270,296.855,-75.862,-177.953,10.413,149.539
C02471=1124.274,296.607,-75.832,-177.956,10.411,149.539
C02472=1124.278,296.359,-75.800,-177.960,10.408,149.539
C02473=1124.283,296.111,-75.769,-177.962,10.405,149.540
C02474=1124.286,295.863,-75.737,-177.966,10.403,149.540
C02475=1124.291,295.615,-75.706,-177.969,10.400,149.540
C02476=1124.295,295.367,-75.675,-177.972,10.398,149.540
C02477=1124.299,295.119,-75.643,-177.975,10.395,149.540
C02478=1124.302,294.906,-75.616,-177.977,10.393,149.540
C02479=1124.306,294.693,-75.590,-177.980,10.391,149.541
C02480=1124.309,294.480,-75.563,-177.983,10.389,149.541
C02481=1124.313,294.267,-75.536,-177.985,10.387,149.541
C02482=1124.316,294.053,-75.509,-177.988,10.385,149.541
C02483=1124.320,293.840,-75.482,-177.991,10.382,149.541
C02484=1124.323,293.626,-75.455,-177.993,10.380,149.541
C02485=1124.327,293.414,-75.428,-177.996,10.377,149.541
C02486=1124.331,293.166,-75.397,-177.999,10.376,149.542
C02487=1124.335,292.917,-75.366,-178.002,10.373,149.542
C02488=1124.340,292.670,-75.335,-178.005,10.371,149.542
C02489=1124.344,292.421,-75.304,-178.008,10.368,149.542
C02490=1124.347,292.174,-75.273,-178.011,10.365,149.542
C02491=1124.351,291.926,-75.242,-178.014,10.363,149.543
C02492=1124.356,291.678,-75.211,-178.018,10.360,149.543
C02493=1124.360,291.430,-75.179,-178.021,10.357,149.543
C02494=1124.364,291.182,-75.148,-178.024,10.355,149.543
C02495=1124.368,290.933,-75.117,-178.027,10.352,149.543
C02496=1124.372,290.686,-75.086,-178.030,10.349,149.543
C02497=1124.376,290.438,-75.056,-178.032,10.348,149.544
C02498=1124.380,290.189,-75.024,-178.035,10.345,149.544
C02499=1124.385,289.941,-74.994,-178.039,10.343,149.544
C02500=1124.389,289.693,-74.962,-178.042,10.340,149.544
C02501=1124.393,289.446,-74.932,-178.045,10.337,149.544
C02502=1124.397,289.197,-74.900,-178.048,10.335,149.544
C02503=1124.401,288.949,-74.870,-178.051,10.332,149.545
C02504=1124.406,288.701,-74.839,-178.054,10.330,149.545
C02505=1124.410,288.452,-74.808,-178.058,10.327,149.545
C02506=1124.413,288.205,-74.777,-178.061,10.324,149.545
C02507=1124.418,287.958,-74.746,-178.063,10.322,149.545
C02508=1124.422,287.709,-74.715,-178.066,10.320,149.546
C02509=1124.426,287.461,-74.685,-178.069,10.317,149.546
C02510=1124.430,287.213,-74.654,-178.072,10.315,149.546
C02511=1124.435,286.965,-74.623,-178.075,10.312,149.546
C02512=1124.439,286.717,-74.592,-178.079,10.310,149.546
C02513=1124.442,286.468,-74.562,-178.082,10.307,149.546
C02514=1124.447,286.220,-74.531,-178.085,10.304,149.547
C02515=1124.452,285.972,-74.500,-178.088,10.302,149.547
C02516=1124.455,285.724,-74.470,-178.091,10.299,149.547
C02517=1124.460,285.476,-74.439,-178.094,10.297,149.547
C02518=1124.464,285.228,-74.408,-178.097,10.294,149.547
C02519=1124.467,284.980,-74.378,-178.100,10.292,149.548
C02520=1124.472,284.732,-74.347,-178.103,10.289,149.548
C02521=1124.476,284.484,-74.317,-178.106,10.287,149.548
C02522=1124.481,284.236,-74.286,-178.109,10.284,149.548
C02523=1124.485,283.988,-74.255,-178.112,10.281,149.548
C02524=1124.488,283.740,-74.225,-178.115,10.279,149.548
C02525=1124.493,283.492,-74.194,-178.118,10.276,149.548
C02526=1124.497,283.244,-74.164,-178.122,10.274,149.549
C02527=1124.501,282.995,-74.133,-178.124,10.272,149.549
C02528=1124.506,282.747,-74.102,-178.127,10.269,149.549
C02529=1124.510,282.499,-74.072,-178.130,10.267,149.549
C02530=1124.514,282.251,-74.042,-178.133,10.264,149.549
C02531=1124.518,282.003,-74.011,-178.136,10.261,149.550
C02532=1124.522,281.755,-73.980,-178.139,10.259,149.550
C02533=1124.526,281.507,-73.951,-178.143,10.256,149.550
C02534=1124.530,281.294,-73.924,-178.146,10.253,149.550
C02535=1124.533,281.080,-73.898,-178.148,10.252,149.550
C02536=1124.537,280.867,-73.872,-178.151,10.249,149.551
C02537=1124.541,280.654,-73.846,-178.154,10.246,149.551
C02538=1124.545,280.441,-73.820,-178.157,10.245,149.551
C02539=1124.548,280.228,-73.794,-178.160,10.242,149.551
C02540=1124.552,280.013,-73.768,-178.163,10.240,149.551
C02541=1124.555,279.801,-73.742,-178.166,10.238,149.551
C02542=1124.560,279.552,-73.712,-178.170,10.234,149.552
C02543=1124.564,279.304,-73.682,-178.173,10.232,149.552
C02544=1124.568,279.056,-73.651,-178.176,10.229,149.552
C02545=1124.572,278.807,-73.621,-178.179,10.226,149.552
C02546=1124.576,278.560,-73.591,-178.183,10.223,149.552
C02547=1124.580,278.312,-73.560,-178.186,10.220,149.553
C02548=1124.585,278.064,-73.531,-178.189,10.218,149.553
C02549=1124.589,277.816,-73.500,-178.192,10.215,149.553
C02550=1124.593,277.567,-73.471,-178.195,10.213,149.553
C02551=1124.597,277.320,-73.440,-178.199,10.209,149.553
C02552=1124.602,277.070,-73.410,-178.202,10.207,149.553
C02553=1124.605,276.823,-73.380,-178.205,10.204,149.553
C02554=1124.610,276.574,-73.350,-178.208,10.201,149.554
C02555=1124.613,276.327,-73.320,-178.211,10.199,149.554
C02556=1124.618,276.078,-73.290,-178.214,10.196,149.554
C02557=1124.623,275.830,-73.261,-178.217,10.193,149.554
C02558=1124.626,275.582,-73.230,-178.220,10.191,149.554
C02559=1124.631,275.334,-73.200,-178.223,10.188,149.554
C02560=1124.635,275.086,-73.170,-178.226,10.185,149.555
C02561=1124.639,274.837,-73.140,-178.230,10.183,149.555
C02562=1124.643,274.589,-73.111,-178.232,10.180,149.555
C02563=1124.648,274.341,-73.080,-178.235,10.177,149.555
C02564=1124.652,274.093,-73.051,-178.238,10.174,149.555
C02565=1124.656,273.844,-73.021,-178.241,10.172,149.555
C02566=1124.660,273.597,-72.991,-178.245,10.169,149.556
C02567=1124.664,273.348,-72.962,-178.248,10.167,149.556
C02568=1124.669,273.100,-72.932,-178.251,10.164,149.556
C02569=1124.673,272.852,-72.901,-178.253,10.161,149.556
C02570=1124.677,272.604,-72.872,-178.256,10.158,149.556
C02571=1124.681,272.356,-72.843,-178.259,10.156,149.556
C02572=1124.685,272.107,-72.813,-178.262,10.153,149.556
C02573=1124.690,271.859,-72.784,-178.265,10.150,149.556
C02574=1124.694,271.611,-72.753,-178.268,10.147,149.556
C02575=1124.698,271.363,-72.723,-178.270,10.145,149.556
C02576=1124.703,271.115,-72.694,-178.274,10.143,149.557
C02577=1124.707,270.866,-72.665,-178.277,10.140,149.557
C02578=1124.711,270.618,-72.635,-178.280,10.137,149.557
C02579=1124.715,270.370,-72.606,-178.283,10.135,149.557
C02580=1124.719,270.122,-72.575,-178.285,10.133,149.557
C02581=1124.723,269.874,-72.546,-178.288,10.130,149.557
C02582=1124.727,269.626,-72.517,-178.291,10.127,149.557
C02583=1124.731,269.377,-72.487,-178.294,10.124,149.557
C02584=1124.736,269.129,-72.458,-178.296,10.122,149.558
C02585=1124.741,268.881,-72.428,-178.299,10.119,149.557
C02586=1124.745,268.632,-72.398,-178.301,10.116,149.558
C02587=1124.749,268.384,-72.369,-178.304,10.114,149.558
C02588=1124.753,268.136,-72.339,-178.307,10.112,149.558
C02589=1124.757,267.888,-72.310,-178.310,10.109,149.558
C02590=1124.761,267.674,-72.285,-178.312,10.107,149.558
C02591=1124.764,267.461,-72.259,-178.314,10.105,149.558
C02592=1124.768,267.247,-72.234,-178.317,10.103,149.558
C02593=1124.772,267.035,-72.209,-178.319,10.101,149.558
C02594=1124.776,266.821,-72.184,-178.321,10.099,149.558
C02595=1124.779,266.608,-72.159,-178.323,10.097,149.558
C02596=1124.783,266.394,-72.134,-178.325,10.095,149.559
C02597=1124.787,266.181,-72.108,-178.328,10.093,149.559
C02598=1124.791,265.932,-72.079,-178.331,10.090,149.559
C02599=1124.795,265.684,-72.050,-178.333,10.088,149.559
C02600=1124.799,265.436,-72.020,-178.336,10.085,149.559
C02601=1124.803,265.188,-71.991,-178.338,10.083,149.559
C02602=1124.808,264.939,-71.962,-178.340,10.081,149.559
C02603=1124.812,264.691,-71.933,-178.343,10.078,149.559
C02604=1124.817,264.443,-71.904,-178.345,10.076,149.559
C02605=1124.821,264.195,-71.874,-178.349,10.073,149.560
C02606=1124.825,263.947,-71.845,-178.353,10.070,149.560
C02607=1124.829,263.698,-71.816,-178.356,10.067,149.560
C02608=1124.834,263.449,-71.787,-178.360,10.064,149.560
C02609=1124.838,263.201,-71.757,-178.364,10.060,149.560
C02610=1124.842,262.954,-71.729,-178.367,10.058,149.561
C02611=1124.846,262.705,-71.700,-178.371,10.055,149.561
C02612=1124.851,262.457,-71.670,-178.374,10.052,149.561
C02613=1124.855,262.208,-71.641,-178.378,10.049,149.561
C02614=1124.859,261.960,-71.612,-178.382,10.045,149.561
C02615=1124.864,261.712,-71.583,-178.385,10.043,149.562
C02616=1124.867,261.464,-71.554,-178.388,10.040,149.562
C02617=1124.872,261.215,-71.525,-178.392,10.037,149.562
C02618=1124.876,260.967,-71.496,-178.394,10.034,149.562
C02619=1124.880,260.719,-71.467,-178.398,10.031,149.562
C02620=1124.885,260.471,-71.439,-178.401,10.028,149.562
C02621=1124.889,260.222,-71.409,-178.405,10.024,149.563
C02622=1124.893,259.974,-71.381,-178.408,10.022,149.563
C02623=1124.897,259.725,-71.351,-178.411,10.019,149.563
C02624=1124.902,259.477,-71.323,-178.414,10.016,149.563
C02625=1124.906,259.229,-71.294,-178.417,10.013,149.563
C02626=1124.910,258.980,-71.265,-178.421,10.010,149.563
C02627=1124.914,258.732,-71.236,-178.424,10.007,149.563
C02628=1124.919,258.484,-71.208,-178.427,10.005,149.563
C02629=1124.923,258.236,-71.179,-178.430,10.001,149.564
C02630=1124.927,257.987,-71.150,-178.433,9.998,149.563
C02631=1124.932,257.739,-71.122,-178.436,9.995,149.564
C02632=1124.936,257.491,-71.093,-178.439,9.993,149.564
C02633=1124.940,257.242,-71.064,-178.442,9.990,149.564
C02634=1124.945,256.995,-71.035,-178.445,9.987,149.564
C02635=1124.948,256.746,-71.007,-178.447,9.984,149.564
C02636=1124.953,256.497,-70.978,-178.450,9.982,149.564
C02637=1124.958,256.250,-70.949,-178.453,9.978,149.564
C02638=1124.962,256.001,-70.921,-178.456,9.976,149.564
C02639=1124.966,255.752,-70.892,-178.456,9.975,149.564
C02640=1124.970,255.504,-70.865,-178.456,9.973,149.564
C02641=1124.975,255.256,-70.835,-178.457,9.972,149.564
C02642=1124.978,255.007,-70.807,-178.457,9.971,149.563
C02643=1124.983,254.759,-70.779,-178.458,9.969,149.563
C02644=1124.988,254.511,-70.749,-178.458,9.968,149.563
C02645=1124.991,254.262,-70.721,-178.459,9.967,149.563
C02646=1124.996,254.049,-70.697,-178.461,9.965,149.563
C02647=1124.999,253.836,-70.672,-178.462,9.964,149.563
C02648=1125.002,253.622,-70.648,-178.463,9.962,149.563
C02649=1125.006,253.409,-70.623,-178.465,9.961,149.563
C02650=1125.010,253.194,-70.598,-178.466,9.959,149.563
C02651=1125.014,252.981,-70.574,-178.468,9.957,149.563
C02652=1125.017,252.768,-70.550,-178.470,9.955,149.563
C02653=1125.021,252.554,-70.525,-178.472,9.954,149.563
C02654=1125.026,252.306,-70.497,-178.475,9.951,149.563
C02655=1125.030,252.058,-70.468,-178.478,9.948,149.563
C02656=1125.034,251.809,-70.439,-178.481,9.946,149.564
C02657=1125.038,251.561,-70.411,-178.484,9.943,149.564
C02658=1125.042,251.313,-70.383,-178.488,9.941,149.564
C02659=1125.047,251.064,-70.355,-178.492,9.938,149.564
C02660=1125.051,250.816,-70.327,-178.496,9.935,149.565
C02661=1125.056,250.567,-70.298,-178.500,9.931,149.565
C02662=1125.060,250.320,-70.270,-178.504,9.928,149.565
C02663=1125.064,250.071,-70.241,-178.508,9.924,149.566
C02664=1125.068,249.823,-70.213,-178.513,9.921,149.566
C02665=1125.072,249.574,-70.185,-178.518,9.917,149.566
C02666=1125.077,249.326,-70.157,-178.523,9.913,149.567
C02667=1125.081,249.078,-70.128,-178.528,9.909,149.567
C02668=1125.086,248.829,-70.100,-178.533,9.905,149.568
C02669=1125.090,248.581,-70.072,-178.539,9.900,149.568
C02670=1125.094,248.332,-70.045,-178.545,9.896,149.568
C02671=1125.098,248.084,-70.017,-178.551,9.891,149.569
C02672=1125.103,247.836,-69.988,-178.557,9.887,149.569
C02673=1125.107,247.587,-69.960,-178.563,9.881,149.570
C02674=1125.111,247.339,-69.932,-178.567,9.878,149.570
C02675=1125.116,247.090,-69.904,-178.569,9.875,149.570
C02676=1125.121,246.842,-69.877,-178.570,9.873,149.570
C02677=1125.124,246.593,-69.848,-178.572,9.871,149.569
C02678=1125.129,246.345,-69.821,-178.574,9.868,149.569
C02679=1125.132,246.097,-69.792,-178.574,9.866,149.569
C02680=1125.138,245.848,-69.765,-178.576,9.864,149.569
C02681=1125.142,245.600,-69.737,-178.578,9.862,149.569
C02682=1125.146,245.351,-69.709,-178.580,9.859,149.569
C02683=1125.150,245.104,-69.681,-178.582,9.857,149.569
C02684=1125.154,244.854,-69.654,-178.583,9.855,149.569
C02685=1125.159,244.606,-69.625,-178.585,9.853,149.569
C02686=1125.164,244.358,-69.598,-178.587,9.850,149.569
C02687=1125.168,244.109,-69.570,-178.589,9.848,149.569
C02688=1125.172,243.861,-69.542,-178.590,9.846,149.568
C02689=1125.176,243.613,-69.514,-178.592,9.843,149.568
C02690=1125.181,243.364,-69.487,-178.594,9.841,149.568
C02691=1125.186,243.116,-69.459,-178.596,9.839,149.568
C02692=1125.189,242.867,-69.431,-178.598,9.836,149.568
C02693=1125.194,242.619,-69.404,-178.600,9.834,149.568
C02694=1125.198,242.370,-69.375,-178.602,9.832,149.568
C02695=1125.202,242.122,-69.348,-178.604,9.830,149.568
C02696=1125.207,241.874,-69.321,-178.607,9.827,149.568
C02697=1125.211,241.625,-69.292,-178.609,9.825,149.568
C02698=1125.215,241.377,-69.265,-178.611,9.822,149.568
C02699=1125.220,241.129,-69.237,-178.613,9.820,149.568
C02700=1125.224,240.879,-69.210,-178.615,9.818,149.568
C02701=1125.229,240.632,-69.182,-178.618,9.815,149.568
C02702=1125.232,240.418,-69.158,-178.620,9.813,149.568
C02703=1125.236,240.204,-69.135,-178.621,9.811,149.568
C02704=1125.240,239.990,-69.111,-178.623,9.809,149.568
C02705=1125.244,239.777,-69.087,-178.625,9.807,149.568
C02706=1125.247,239.563,-69.064,-178.627,9.805,149.568
C02707=1125.251,239.349,-69.040,-178.630,9.803,149.569
C02708=1125.255,239.136,-69.016,-178.632,9.801,149.569
C02709=1125.258,238.923,-68.993,-178.634,9.798,149.569
C02710=1125.262,238.673,-68.965,-178.637,9.796,149.569
C02711=1125.267,238.425,-68.938,-178.639,9.793,149.569
C02712=1125.271,238.177,-68.910,-178.642,9.791,149.569
C02713=1125.275,237.928,-68.883,-178.645,9.788,149.569
C02714=1125.280,237.680,-68.855,-178.647,9.786,149.569
C02715=1125.284,237.432,-68.828,-178.649,9.783,149.569
C02716=1125.288,237.182,-68.801,-178.652,9.780,149.569
C02717=1125.293,236.934,-68.773,-178.655,9.778,149.569
C02718=1125.297,236.686,-68.746,-178.658,9.775,149.569
C02719=1125.302,236.437,-68.719,-178.661,9.773,149.570
C02720=1125.306,236.189,-68.691,-178.663,9.770,149.570
C02721=1125.311,235.940,-68.663,-178.666,9.767,149.570
C02722=1125.315,235.692,-68.636,-178.669,9.764,149.570
C02723=1125.320,235.444,-68.609,-178.672,9.761,149.570
C02724=1125.324,235.195,-68.581,-178.675,9.759,149.570
C02725=1125.328,234.946,-68.554,-178.678,9.756,149.570
C02726=1125.333,234.698,-68.527,-178.681,9.753,149.570
C02727=1125.337,234.450,-68.500,-178.684,9.750,149.570
C02728=1125.341,234.201,-68.472,-178.687,9.748,149.570
C02729=1125.345,233.953,-68.445,-178.690,9.745,149.571
C02730=1125.350,233.704,-68.418,-178.693,9.742,149.571
C02731=1125.355,233.456,-68.391,-178.696,9.739,149.571
C02732=1125.359,233.207,-68.364,-178.699,9.736,149.571
C02733=1125.362,232.959,-68.337,-178.702,9.733,149.571
C02734=1125.367,232.710,-68.310,-178.706,9.730,149.571
C02735=1125.372,232.462,-68.283,-178.709,9.727,149.572
C02736=1125.376,232.213,-68.256,-178.712,9.724,149.572
C02737=1125.381,231.965,-68.228,-178.715,9.721,149.572
C02738=1125.385,231.717,-68.202,-178.718,9.718,149.572
C02739=1125.389,231.467,-68.175,-178.722,9.715,149.572
C02740=1125.393,231.219,-68.147,-178.725,9.712,149.572
C02741=1125.398,230.970,-68.120,-178.729,9.708,149.572
C02742=1125.402,230.722,-68.094,-178.732,9.705,149.572
C02743=1125.407,230.474,-68.067,-178.735,9.702,149.573
C02744=1125.411,230.225,-68.040,-178.739,9.699,149.573
C02745=1125.415,229.977,-68.013,-178.743,9.695,149.573
C02746=1125.420,229.729,-67.986,-178.746,9.692,149.573
C02747=1125.425,229.480,-67.959,-178.750,9.688,149.573
C02748=1125.428,229.231,-67.932,-178.753,9.685,149.573
C02749=1125.433,228.983,-67.905,-178.756,9.682,149.573
C02750=1125.438,228.734,-67.879,-178.760,9.679,149.574
C02751=1125.441,228.485,-67.853,-178.763,9.675,149.574
C02752=1125.446,228.237,-67.825,-178.767,9.671,149.574
C02753=1125.451,227.988,-67.798,-178.770,9.669,149.574
C02754=1125.455,227.740,-67.772,-178.773,9.665,149.574
C02755=1125.459,227.492,-67.745,-178.777,9.661,149.574
C02756=1125.464,227.243,-67.719,-178.780,9.659,149.574
C02757=1125.468,226.994,-67.692,-178.783,9.655,149.574
C02758=1125.472,226.781,-67.669,-178.786,9.652,149.574
C02759=1125.476,226.566,-67.646,-178.789,9.649,149.574
C02760=1125.480,226.353,-67.623,-178.791,9.646,149.574
C02761=1125.484,226.139,-67.601,-178.794,9.643,149.574
C02762=1125.486,225.925,-67.578,-178.797,9.640,149.574
C02763=1125.491,225.711,-67.555,-178.800,9.637,149.574
C02764=1125.495,225.498,-67.532,-178.802,9.635,149.574
C02765=1125.499,225.284,-67.510,-178.804,9.632,149.574
C02766=1125.503,225.036,-67.483,-178.808,9.629,149.574
C02767=1125.508,224.787,-67.457,-178.810,9.625,149.574
C02768=1125.512,224.538,-67.430,-178.814,9.622,149.574
C02769=1125.516,224.290,-67.403,-178.816,9.619,149.574
C02770=1125.520,224.041,-67.378,-178.819,9.616,149.574
C02771=1125.525,223.793,-67.350,-178.822,9.612,149.574
C02772=1125.529,223.544,-67.325,-178.825,9.609,149.574
C02773=1125.534,223.296,-67.298,-178.828,9.606,149.574
C02774=1125.538,223.047,-67.272,-178.831,9.602,149.574
C02775=1125.543,222.798,-67.245,-178.833,9.599,149.574
C02776=1125.547,222.549,-67.219,-178.836,9.596,149.574
C02777=1125.551,222.301,-67.193,-178.839,9.593,149.574
C02778=1125.556,222.052,-67.166,-178.842,9.589,149.574
C02779=1125.560,221.804,-67.140,-178.844,9.586,149.574
C02780=1125.565,221.556,-67.114,-178.847,9.583,149.574
C02781=1125.569,221.307,-67.087,-178.849,9.580,149.574
C02782=1125.573,221.059,-67.062,-178.852,9.577,149.574
C02783=1125.578,220.809,-67.035,-178.854,9.574,149.574
C02784=1125.582,220.561,-67.009,-178.857,9.571,149.574
C02785=1125.587,220.312,-66.983,-178.860,9.567,149.574
C02786=1125.592,220.063,-66.957,-178.862,9.564,149.574
C02787=1125.595,219.815,-66.930,-178.865,9.561,149.574
C02788=1125.600,219.567,-66.905,-178.867,9.558,149.573
C02789=1125.604,219.318,-66.879,-178.869,9.555,149.573
C02790=1125.609,219.070,-66.852,-178.872,9.552,149.573
C02791=1125.613,218.821,-66.826,-178.874,9.548,149.573
C02792=1125.618,218.572,-66.801,-178.877,9.545,149.573
C02793=1125.622,218.324,-66.774,-178.878,9.543,149.573
C02794=1125.626,218.075,-66.748,-178.881,9.540,149.573
C02795=1125.631,217.827,-66.722,-178.883,9.536,149.573
C02796=1125.636,217.578,-66.697,-178.886,9.533,149.573
C02797=1125.640,217.329,-66.671,-178.887,9.531,149.572
C02798=1125.644,217.081,-66.644,-178.890,9.528,149.572
C02799=1125.649,216.832,-66.618,-178.892,9.524,149.572
C02800=1125.653,216.584,-66.593,-178.894,9.522,149.572
C02801=1125.658,216.335,-66.567,-178.896,9.519,149.572
C02802=1125.662,216.086,-66.541,-178.898,9.516,149.572
C02803=1125.666,215.838,-66.515,-178.900,9.513,149.572
C02804=1125.671,215.589,-66.488,-178.902,9.510,149.572
C02805=1125.676,215.341,-66.463,-178.905,9.507,149.572
C02806=1125.680,215.092,-66.437,-178.906,9.505,149.571
C02807=1125.684,214.843,-66.411,-178.909,9.502,149.571
C02808=1125.688,214.594,-66.386,-178.910,9.499,149.571
C02809=1125.693,214.346,-66.360,-178.912,9.497,149.571
C02810=1125.697,214.097,-66.335,-178.914,9.493,149.571
C02811=1125.702,213.849,-66.309,-178.916,9.491,149.571
C02812=1125.707,213.599,-66.282,-178.918,9.488,149.571
C02813=1125.711,213.351,-66.257,-178.920,9.486,149.570
C02814=1125.714,213.137,-66.235,-178.921,9.483,149.570
C02815=1125.718,212.923,-66.212,-178.923,9.481,149.570
C02816=1125.722,212.710,-66.190,-178.925,9.478,149.570
C02817=1125.726,212.495,-66.168,-178.927,9.476,149.570
C02818=1125.730,212.282,-66.147,-178.928,9.474,149.570
C02819=1125.734,212.068,-66.124,-178.929,9.472,149.570
C02820=1125.737,211.854,-66.102,-178.931,9.469,149.570
C02821=1125.741,211.640,-66.080,-178.933,9.467,149.570
C02822=1125.746,211.391,-66.054,-178.935,9.465,149.570
C02823=1125.751,211.143,-66.029,-178.938,9.462,149.569
C02824=1125.755,210.894,-66.003,-178.940,9.459,149.569
C02825=1125.759,210.645,-65.978,-178.941,9.457,149.569
C02826=1125.763,210.396,-65.952,-178.944,9.454,149.569
C02827=1125.768,210.148,-65.927,-178.946,9.452,149.569
C02828=1125.772,209.899,-65.901,-178.948,9.448,149.569
C02829=1125.777,209.651,-65.875,-178.950,9.446,149.569
C02830=1125.781,209.402,-65.850,-178.953,9.443,149.569
C02831=1125.786,209.154,-65.824,-178.956,9.440,149.569
C02832=1125.790,208.904,-65.799,-178.958,9.438,149.569
C02833=1125.795,208.656,-65.774,-178.960,9.435,149.569
C02834=1125.799,208.407,-65.748,-178.962,9.433,149.569
C02835=1125.804,208.159,-65.722,-178.965,9.430,149.569
C02836=1125.808,207.910,-65.697,-178.968,9.427,149.569
C02837=1125.813,207.661,-65.672,-178.970,9.424,149.569
C02838=1125.818,207.413,-65.646,-178.972,9.422,149.569
C02839=1125.822,207.164,-65.620,-178.975,9.419,149.569
C02840=1125.826,206.915,-65.595,-178.978,9.416,149.569
C02841=1125.831,206.667,-65.571,-178.981,9.413,149.570
C02842=1125.835,206.418,-65.545,-178.984,9.410,149.570
C02843=1125.840,206.170,-65.520,-178.986,9.407,149.570
C02844=1125.844,205.921,-65.494,-178.989,9.405,149.570
C02845=1125.848,205.672,-65.469,-178.992,9.402,149.570
C02846=1125.853,205.424,-65.443,-178.994,9.399,149.570
C02847=1125.858,205.174,-65.418,-178.997,9.397,149.570
C02848=1125.863,204.926,-65.393,-179.001,9.393,149.570
C02849=1125.866,204.678,-65.368,-179.003,9.390,149.570
C02850=1125.871,204.429,-65.343,-179.006,9.387,149.570
C02851=1125.875,204.180,-65.317,-179.009,9.384,149.570
C02852=1125.881,203.931,-65.293,-179.012,9.382,149.571
C02853=1125.885,203.683,-65.267,-179.015,9.379,149.571
C02854=1125.888,203.434,-65.242,-179.019,9.375,149.571
C02855=1125.893,203.185,-65.217,-179.021,9.372,149.571
C02856=1125.898,202.937,-65.191,-179.024,9.370,149.571
C02857=1125.903,202.688,-65.167,-179.027,9.367,149.571
C02858=1125.906,202.439,-65.142,-179.031,9.363,149.571
C02859=1125.911,202.191,-65.117,-179.034,9.361,149.571
C02860=1125.916,201.942,-65.091,-179.037,9.357,149.572
C02861=1125.921,201.693,-65.066,-179.040,9.354,149.572
C02862=1125.924,201.444,-65.042,-179.044,9.351,149.572
C02863=1125.929,201.196,-65.017,-179.047,9.348,149.572
C02864=1125.934,200.946,-64.992,-179.050,9.345,149.572
C02865=1125.938,200.699,-64.967,-179.053,9.342,149.572
C02866=1125.942,200.449,-64.942,-179.056,9.338,149.572
C02867=1125.948,200.201,-64.917,-179.060,9.334,149.572
C02868=1125.951,199.952,-64.892,-179.063,9.331,149.572
C02869=1125.956,199.703,-64.867,-179.066,9.328,149.573
C02870=1125.960,199.489,-64.846,-179.069,9.325,149.573
C02871=1125.963,199.275,-64.824,-179.073,9.322,149.573
C02872=1125.967,199.061,-64.804,-179.076,9.319,149.573
C02873=1125.972,198.848,-64.782,-179.079,9.316,149.573
C02874=1125.976,198.633,-64.760,-179.081,9.313,149.573
C02875=1125.980,198.419,-64.739,-179.085,9.310,149.573
C02876=1125.983,198.205,-64.718,-179.088,9.307,149.573
C02877=1125.987,197.991,-64.697,-179.091,9.304,149.574
C02878=1125.991,197.742,-64.673,-179.094,9.301,149.574
C02879=1125.996,197.493,-64.648,-179.098,9.297,149.574
C02880=1126.000,197.245,-64.623,-179.102,9.293,149.574
C02881=1126.005,196.996,-64.598,-179.105,9.289,149.574
C02882=1126.009,196.747,-64.574,-179.109,9.286,149.574
C02883=1126.014,196.499,-64.549,-179.113,9.282,149.574
C02884=1126.018,196.250,-64.525,-179.116,9.279,149.574
C02885=1126.023,196.001,-64.500,-179.118,9.276,149.574
C02886=1126.027,195.752,-64.476,-179.119,9.273,149.574
C02887=1126.033,195.504,-64.451,-179.121,9.271,149.574
C02888=1126.036,195.254,-64.427,-179.122,9.268,149.574
C02889=1126.041,195.006,-64.402,-179.124,9.266,149.574
C02890=1126.046,194.757,-64.378,-179.126,9.263,149.573
C02891=1126.050,194.508,-64.353,-179.127,9.260,149.573
C02892=1126.055,194.260,-64.329,-179.129,9.258,149.573
C02893=1126.059,194.011,-64.305,-179.131,9.255,149.573
C02894=1126.064,193.762,-64.280,-179.133,9.252,149.573
C02895=1126.068,193.513,-64.256,-179.135,9.250,149.573
C02896=1126.073,193.265,-64.231,-179.137,9.247,149.572
C02897=1126.078,193.016,-64.207,-179.138,9.245,149.572
C02898=1126.081,192.767,-64.182,-179.140,9.242,149.572
C02899=1126.087,192.518,-64.158,-179.142,9.240,149.572
C02900=1126.091,192.270,-64.134,-179.144,9.237,149.572
C02901=1126.095,192.020,-64.109,-179.146,9.234,149.572
C02902=1126.100,191.772,-64.085,-179.148,9.232,149.572
C02903=1126.104,191.524,-64.061,-179.150,9.229,149.572
C02904=1126.110,191.274,-64.037,-179.152,9.226,149.572
C02905=1126.114,191.025,-64.012,-179.154,9.224,149.572
C02906=1126.118,190.777,-63.988,-179.156,9.221,149.571
C02907=1126.123,190.528,-63.963,-179.158,9.218,149.571
C02908=1126.127,190.280,-63.939,-179.160,9.216,149.571
C02909=1126.131,190.031,-63.915,-179.162,9.213,149.571
C02910=1126.137,189.781,-63.891,-179.164,9.210,149.571
C02911=1126.141,189.533,-63.867,-179.167,9.207,149.571
C02912=1126.145,189.284,-63.843,-179.169,9.205,149.571
C02913=1126.150,189.036,-63.819,-179.171,9.202,149.571
C02914=1126.154,188.786,-63.794,-179.173,9.200,149.571
C02915=1126.159,188.537,-63.770,-179.176,9.196,149.571
C02916=1126.163,188.289,-63.746,-179.178,9.193,149.571
C02917=1126.169,188.040,-63.722,-179.180,9.191,149.571
C02918=1126.173,187.792,-63.697,-179.183,9.188,149.571
C02919=1126.177,187.542,-63.674,-179.185,9.185,149.571
C02920=1126.181,187.294,-63.650,-179.187,9.182,149.571
C02921=1126.186,187.045,-63.626,-179.190,9.179,149.571
C02922=1126.191,186.796,-63.602,-179.192,9.176,149.571
C02923=1126.196,186.548,-63.578,-179.195,9.173,149.571
C02924=1126.200,186.299,-63.553,-179.196,9.171,149.571
C02925=1126.204,186.049,-63.530,-179.199,9.168,149.571
C02926=1126.209,185.836,-63.509,-179.201,9.166,149.571
C02927=1126.212,185.622,-63.488,-179.204,9.163,149.571
C02928=1126.216,185.407,-63.467,-179.206,9.160,149.571
C02929=1126.220,185.193,-63.447,-179.208,9.157,149.571
C02930=1126.224,184.979,-63.427,-179.210,9.155,149.571
C02931=1126.228,184.765,-63.406,-179.212,9.153,149.571
C02932=1126.232,184.550,-63.385,-179.215,9.149,149.571
C02933=1126.236,184.336,-63.365,-179.217,9.147,149.571
C02934=1126.240,184.088,-63.341,-179.219,9.144,149.571
C02935=1126.245,183.838,-63.317,-179.222,9.141,149.571
C02936=1126.250,183.590,-63.293,-179.224,9.138,149.571
C02937=1126.254,183.341,-63.270,-179.227,9.135,149.571
C02938=1126.259,183.093,-63.246,-179.231,9.132,149.571
C02939=1126.264,182.844,-63.222,-179.233,9.128,149.571
C02940=1126.268,182.595,-63.198,-179.236,9.125,149.571
C02941=1126.273,182.346,-63.175,-179.238,9.122,149.571
C02942=1126.276,182.097,-63.150,-179.241,9.119,149.571
C02943=1126.281,181.848,-63.127,-179.244,9.116,149.571
C02944=1126.286,181.600,-63.103,-179.247,9.112,149.571
C02945=1126.290,181.350,-63.080,-179.249,9.109,149.571
C02946=1126.295,181.101,-63.056,-179.253,9.106,149.571
C02947=1126.299,180.853,-63.032,-179.255,9.103,149.571
C02948=1126.304,180.604,-63.009,-179.258,9.100,149.571
C02949=1126.309,180.355,-62.986,-179.262,9.096,149.571
C02950=1126.313,180.107,-62.961,-179.264,9.093,149.571
C02951=1126.318,179.858,-62.938,-179.267,9.089,149.571
C02952=1126.323,179.608,-62.915,-179.270,9.086,149.571
C02953=1126.327,179.360,-62.891,-179.273,9.082,149.571
C02954=1126.332,179.111,-62.867,-179.276,9.079,149.571
C02955=1126.336,178.862,-62.844,-179.277,9.077,149.571
C02956=1126.341,178.613,-62.821,-179.280,9.074,149.571
C02957=1126.345,178.364,-62.798,-179.282,9.070,149.571
C02958=1126.349,178.116,-62.774,-179.284,9.068,149.570
C02959=1126.354,177.867,-62.750,-179.286,9.065,149.570
C02960=1126.359,177.618,-62.727,-179.288,9.062,149.570
C02961=1126.363,177.369,-62.704,-179.290,9.059,149.570
C02962=1126.368,177.120,-62.680,-179.293,9.056,149.570
C02963=1126.373,176.871,-62.656,-179.294,9.053,149.570
C02964=1126.377,176.622,-62.633,-179.297,9.050,149.570
C02965=1126.381,176.374,-62.610,-179.299,9.047,149.570
C02966=1126.386,176.125,-62.587,-179.301,9.044,149.570
C02967=1126.391,175.875,-62.563,-179.303,9.041,149.569
C02968=1126.396,175.627,-62.540,-179.306,9.038,149.569
C02969=1126.401,175.378,-62.517,-179.308,9.036,149.569
C02970=1126.405,175.129,-62.494,-179.310,9.032,149.569
C02971=1126.409,174.880,-62.471,-179.312,9.029,149.569
C02972=1126.414,174.631,-62.448,-179.314,9.027,149.569
C02973=1126.419,174.382,-62.424,-179.316,9.023,149.569
C02974=1126.423,174.133,-62.401,-179.319,9.020,149.569
C02975=1126.427,173.885,-62.378,-179.321,9.018,149.569
C02976=1126.432,173.636,-62.355,-179.323,9.015,149.569
C02977=1126.437,173.386,-62.331,-179.325,9.011,149.568
C02978=1126.441,173.137,-62.308,-179.328,9.008,149.568
C02979=1126.446,172.889,-62.286,-179.330,9.006,149.568
C02980=1126.451,172.640,-62.262,-179.332,9.002,149.568
C02981=1126.455,172.391,-62.239,-179.334,8.999,149.568
C02982=1126.459,172.177,-62.219,-179.336,8.997,149.568
C02983=1126.463,171.963,-62.199,-179.338,8.994,149.568
C02984=1126.467,171.749,-62.179,-179.340,8.991,149.568
C02985=1126.471,171.534,-62.160,-179.342,8.989,149.568
C02986=1126.475,171.320,-62.139,-179.344,8.986,149.568
C02987=1126.479,171.105,-62.120,-179.346,8.984,149.568
C02988=1126.482,170.892,-62.100,-179.348,8.981,149.568
C02989=1126.487,170.677,-62.080,-179.350,8.978,149.567
C02990=1126.492,170.428,-62.057,-179.353,8.975,149.567
C02991=1126.496,170.180,-62.034,-179.355,8.972,149.567
C02992=1126.501,169.931,-62.011,-179.357,8.969,149.567
C02993=1126.505,169.682,-61.988,-179.359,8.966,149.567
C02994=1126.510,169.433,-61.966,-179.362,8.963,149.567
C02995=1126.515,169.184,-61.943,-179.364,8.960,149.567
C02996=1126.519,168.935,-61.920,-179.366,8.956,149.567
C02997=1126.524,168.686,-61.896,-179.369,8.953,149.567
C02998=1126.528,168.437,-61.873,-179.371,8.951,149.567
C02999=1126.533,168.188,-61.851,-179.373,8.948,149.567
C03000=1126.538,167.939,-61.828,-179.375,8.944,149.567
C03001=1126.542,167.691,-61.805,-179.378,8.941,149.566
C03002=1126.547,167.441,-61.783,-179.380,8.938,149.566
C03003=1126.551,167.193,-61.760,-179.383,8.935,149.566
C03004=1126.556,166.944,-61.737,-179.385,8.932,149.566
C03005=1126.560,166.695,-61.715,-179.387,8.928,149.566
C03006=1126.565,166.446,-61.691,-179.390,8.925,149.566
C03007=1126.570,166.197,-61.668,-179.392,8.922,149.566
C03008=1126.575,165.948,-61.646,-179.394,8.920,149.566
C03009=1126.579,165.699,-61.623,-179.396,8.916,149.566
C03010=1126.584,165.450,-61.601,-179.399,8.913,149.566
C03011=1126.589,165.201,-61.578,-179.401,8.910,149.566
C03012=1126.593,164.952,-61.555,-179.404,8.907,149.565
C03013=1126.597,164.703,-61.533,-179.406,8.904,149.565
C03014=1126.602,164.455,-61.510,-179.409,8.901,149.565
C03015=1126.607,164.205,-61.488,-179.411,8.897,149.565
C03016=1126.611,163.956,-61.465,-179.413,8.894,149.565
C03017=1126.616,163.708,-61.443,-179.416,8.891,149.565
C03018=1126.621,163.459,-61.420,-179.418,8.888,149.565
C03019=1126.625,163.209,-61.398,-179.420,8.884,149.565
C03020=1126.630,162.961,-61.375,-179.423,8.881,149.565
C03021=1126.635,162.712,-61.353,-179.425,8.878,149.565
C03022=1126.639,162.463,-61.330,-179.427,8.875,149.565
C03023=1126.644,162.214,-61.308,-179.431,8.871,149.565
C03024=1126.649,161.965,-61.286,-179.433,8.868,149.564
C03025=1126.653,161.716,-61.263,-179.435,8.864,149.564
C03026=1126.658,161.467,-61.241,-179.438,8.861,149.564
C03027=1126.662,161.218,-61.218,-179.440,8.858,149.564
C03028=1126.666,160.969,-61.196,-179.443,8.855,149.564
C03029=1126.672,160.720,-61.173,-179.445,8.851,149.564
C03030=1126.676,160.471,-61.151,-179.447,8.848,149.564
C03031=1126.681,160.223,-61.129,-179.450,8.845,149.564
C03032=1126.686,159.973,-61.106,-179.452,8.842,149.564
C03033=1126.690,159.724,-61.084,-179.455,8.838,149.564
C03034=1126.695,159.476,-61.062,-179.458,8.835,149.564
C03035=1126.699,159.226,-61.040,-179.460,8.831,149.563
C03036=1126.705,158.977,-61.018,-179.462,8.828,149.563
C03037=1126.709,158.729,-60.995,-179.464,8.825,149.563
C03038=1126.713,158.514,-60.976,-179.467,8.821,149.563
C03039=1126.717,158.300,-60.957,-179.469,8.818,149.563
C03040=1126.720,158.085,-60.938,-179.471,8.816,149.563
C03041=1126.725,157.871,-60.919,-179.473,8.812,149.563
C03042=1126.729,157.656,-60.900,-179.475,8.810,149.563
C03043=1126.733,157.442,-60.881,-179.478,8.807,149.563
C03044=1126.737,157.228,-60.862,-179.480,8.804,149.562
C03045=1126.741,157.014,-60.842,-179.482,8.801,149.562
C03046=1126.745,156.764,-60.820,-179.485,8.797,149.562
C03047=1126.750,156.516,-60.799,-179.487,8.794,149.562
C03048=1126.754,156.266,-60.777,-179.490,8.791,149.562
C03049=1126.759,156.018,-60.755,-179.492,8.787,149.562
C03050=1126.764,155.768,-60.732,-179.495,8.783,149.562
C03051=1126.769,155.520,-60.711,-179.497,8.780,149.562
C03052=1126.773,155.270,-60.689,-179.499,8.777,149.562
C03053=1126.778,155.022,-60.667,-179.502,8.773,149.561
C03054=1126.782,154.773,-60.644,-179.505,8.769,149.561
C03055=1126.787,154.524,-60.623,-179.507,8.766,149.561
C03056=1126.791,154.275,-60.600,-179.510,8.762,149.561
C03057=1126.796,154.026,-60.579,-179.512,8.759,149.561
C03058=1126.801,153.776,-60.557,-179.514,8.755,149.561
C03059=1126.806,153.527,-60.535,-179.518,8.752,149.561
C03060=1126.811,153.278,-60.513,-179.520,8.748,149.561
C03061=1126.815,153.029,-60.491,-179.523,8.744,149.561
C03062=1126.820,152.781,-60.470,-179.525,8.741,149.560
C03063=1126.825,152.531,-60.448,-179.527,8.738,149.560
C03064=1126.829,152.283,-60.426,-179.530,8.733,149.560
C03065=1126.834,152.033,-60.404,-179.532,8.730,149.560
C03066=1126.839,151.785,-60.382,-179.535,8.726,149.560
C03067=1126.843,151.536,-60.361,-179.537,8.722,149.560
C03068=1126.848,151.286,-60.339,-179.541,8.719,149.559
C03069=1126.853,151.037,-60.318,-179.543,8.715,149.559
C03070=1126.857,150.788,-60.296,-179.546,8.711,149.559
C03071=1126.862,150.539,-60.274,-179.548,8.708,149.559
C03072=1126.867,150.291,-60.252,-179.551,8.703,149.559
C03073=1126.872,150.041,-60.231,-179.553,8.700,149.559
C03074=1126.876,149.792,-60.209,-179.556,8.696,149.558
C03075=1126.881,149.544,-60.187,-179.558,8.693,149.558
C03076=1126.885,149.295,-60.166,-179.561,8.689,149.558
C03077=1126.890,149.045,-60.145,-179.563,8.685,149.558
C03078=1126.895,148.797,-60.123,-179.566,8.681,149.558
C03079=1126.899,148.547,-60.101,-179.569,8.677,149.558
C03080=1126.904,148.298,-60.080,-179.571,8.674,149.557
C03081=1126.909,148.049,-60.059,-179.574,8.670,149.557
C03082=1126.913,147.800,-60.037,-179.576,8.666,149.557
C03083=1126.919,147.551,-60.016,-179.579,8.662,149.557
C03084=1126.923,147.303,-59.995,-179.582,8.658,149.557
C03085=1126.927,147.053,-59.973,-179.584,8.655,149.557
C03086=1126.932,146.804,-59.952,-179.587,8.650,149.557
C03087=1126.937,146.555,-59.930,-179.590,8.646,149.556
C03088=1126.942,146.306,-59.909,-179.592,8.643,149.556
C03089=1126.946,146.057,-59.887,-179.595,8.639,149.556
C03090=1126.951,145.808,-59.867,-179.598,8.634,149.556
C03091=1126.956,145.559,-59.845,-179.600,8.630,149.556
C03092=1126.961,145.310,-59.824,-179.602,8.627,149.555
C03093=1126.964,145.061,-59.802,-179.605,8.622,149.555
C03094=1126.969,144.846,-59.784,-179.607,8.620,149.555
C03095=1126.974,144.632,-59.766,-179.608,8.617,149.554
C03096=1126.978,144.417,-59.748,-179.609,8.614,149.554
C03097=1126.982,144.203,-59.729,-179.611,8.611,149.554
C03098=1126.985,143.989,-59.711,-179.612,8.608,149.554
C03099=1126.990,143.774,-59.693,-179.613,8.605,149.553
C03100=1126.993,143.559,-59.675,-179.614,8.602,149.553
C03101=1126.998,143.345,-59.657,-179.615,8.600,149.553
C03102=1127.003,143.096,-59.635,-179.616,8.596,149.552
C03103=1127.007,142.847,-59.615,-179.619,8.593,149.552
C03104=1127.012,142.597,-59.593,-179.620,8.590,149.552
C03105=1127.016,142.348,-59.572,-179.622,8.586,149.551
C03106=1127.021,142.099,-59.551,-179.623,8.583,149.551
C03107=1127.026,141.851,-59.530,-179.624,8.579,149.550
C03108=1127.031,141.602,-59.509,-179.626,8.577,149.550
C03109=1127.035,141.352,-59.488,-179.627,8.573,149.550
C03110=1127.040,141.103,-59.467,-179.629,8.570,149.550
C03111=1127.045,140.854,-59.445,-179.630,8.566,149.549
C03112=1127.049,140.605,-59.425,-179.632,8.564,149.549
C03113=1127.054,140.356,-59.404,-179.634,8.560,149.548
C03114=1127.059,140.107,-59.383,-179.635,8.557,149.548
C03115=1127.063,139.857,-59.362,-179.637,8.553,149.548
C03116=1127.068,139.608,-59.341,-179.638,8.550,149.548
C03117=1127.073,139.359,-59.320,-179.640,8.547,149.547
C03118=1127.078,139.111,-59.299,-179.641,8.544,149.547
C03119=1127.082,138.862,-59.278,-179.643,8.540,149.547
C03120=1127.087,138.612,-59.257,-179.644,8.537,149.546
C03121=1127.092,138.363,-59.237,-179.646,8.533,149.546
C03122=1127.097,138.114,-59.216,-179.647,8.531,149.546
C03123=1127.100,137.865,-59.194,-179.649,8.527,149.545
C03124=1127.106,137.616,-59.174,-179.650,8.524,149.545
C03125=1127.111,137.367,-59.153,-179.652,8.520,149.545
C03126=1127.115,137.118,-59.132,-179.654,8.517,149.544
C03127=1127.120,136.868,-59.111,-179.656,8.514,149.544
C03128=1127.125,136.620,-59.091,-179.657,8.511,149.544
C03129=1127.130,136.370,-59.070,-179.659,8.507,149.543
C03130=1127.134,136.122,-59.049,-179.660,8.504,149.543
C03131=1127.139,135.873,-59.028,-179.662,8.501,149.543
C03132=1127.144,135.624,-59.007,-179.663,8.497,149.542
C03133=1127.148,135.375,-58.987,-179.665,8.494,149.542
C03134=1127.153,135.126,-58.966,-179.667,8.491,149.542
C03135=1127.157,134.876,-58.945,-179.668,8.488,149.541
C03136=1127.162,134.627,-58.924,-179.670,8.484,149.541
C03137=1127.167,134.378,-58.904,-179.671,8.481,149.541
C03138=1127.172,134.128,-58.883,-179.673,8.478,149.541
C03139=1127.176,133.879,-58.863,-179.675,8.474,149.540
C03140=1127.182,133.630,-58.842,-179.676,8.471,149.540
C03141=1127.186,133.381,-58.821,-179.678,8.468,149.540
C03142=1127.190,133.132,-58.801,-179.680,8.465,149.539
C03143=1127.196,132.883,-58.780,-179.681,8.461,149.539
C03144=1127.200,132.634,-58.760,-179.683,8.458,149.539
C03145=1127.205,132.385,-58.739,-179.685,8.455,149.539
C03146=1127.210,132.136,-58.718,-179.686,8.451,149.538
C03147=1127.214,131.887,-58.698,-179.688,8.448,149.538
C03148=1127.219,131.638,-58.677,-179.690,8.445,149.538
C03149=1127.224,131.389,-58.657,-179.691,8.442,149.537
C03150=1127.228,131.174,-58.640,-179.693,8.438,149.537
C03151=1127.233,130.959,-58.622,-179.694,8.435,149.537
C03152=1127.236,130.745,-58.604,-179.696,8.433,149.537
C03153=1127.240,130.530,-58.587,-179.697,8.430,149.536
C03154=1127.244,130.315,-58.569,-179.699,8.427,149.536
C03155=1127.249,130.101,-58.551,-179.700,8.424,149.536
C03156=1127.253,129.886,-58.534,-179.702,8.422,149.536
C03157=1127.256,129.672,-58.516,-179.703,8.419,149.535
C03158=1127.262,129.422,-58.495,-179.705,8.415,149.535
C03159=1127.266,129.173,-58.475,-179.707,8.412,149.535
C03160=1127.271,128.924,-58.454,-179.708,8.409,149.535
C03161=1127.276,128.676,-58.435,-179.710,8.405,149.534
C03162=1127.281,128.426,-58.414,-179.712,8.402,149.534
C03163=1127.285,128.177,-58.394,-179.713,8.399,149.534
C03164=1127.290,127.928,-58.373,-179.716,8.395,149.534
C03165=1127.295,127.679,-58.354,-179.717,8.392,149.533
C03166=1127.300,127.430,-58.333,-179.719,8.389,149.533
C03167=1127.304,127.181,-58.312,-179.721,8.385,149.533
C03168=1127.309,126.931,-58.293,-179.723,8.382,149.532
C03169=1127.313,126.682,-58.272,-179.724,8.379,149.532
C03170=1127.319,126.433,-58.251,-179.726,8.375,149.532
C03171=1127.323,126.184,-58.231,-179.728,8.372,149.532
C03172=1127.328,125.934,-58.211,-179.729,8.369,149.531
C03173=1127.333,125.686,-58.191,-179.731,8.366,149.531
C03174=1127.337,125.437,-58.171,-179.733,8.362,149.531
C03175=1127.342,125.188,-58.151,-179.734,8.359,149.530
C03176=1127.347,124.938,-58.130,-179.737,8.355,149.530
C03177=1127.352,124.689,-58.111,-179.739,8.352,149.530
C03178=1127.356,124.440,-58.090,-179.740,8.348,149.530
C03179=1127.361,124.191,-58.070,-179.742,8.345,149.529
C03180=1127.366,123.942,-58.051,-179.744,8.342,149.529
C03181=1127.371,123.693,-58.030,-179.746,8.338,149.529
C03182=1127.375,123.444,-58.011,-179.747,8.336,149.529
C03183=1127.381,123.194,-57.990,-179.749,8.332,149.528
C03184=1127.385,122.945,-57.970,-179.751,8.328,149.528
C03185=1127.390,122.696,-57.950,-179.753,8.325,149.528
C03186=1127.395,122.447,-57.930,-179.754,8.322,149.528
C03187=1127.399,122.198,-57.910,-179.756,8.318,149.527
C03188=1127.404,121.948,-57.890,-179.758,8.315,149.527
C03189=1127.409,121.699,-57.870,-179.760,8.311,149.527
C03190=1127.413,121.450,-57.850,-179.762,8.308,149.526
C03191=1127.418,121.202,-57.830,-179.764,8.305,149.526
C03192=1127.423,120.952,-57.811,-179.765,8.301,149.526
C03193=1127.428,120.703,-57.790,-179.767,8.298,149.526
C03194=1127.432,120.453,-57.771,-179.769,8.294,149.525
C03195=1127.437,120.205,-57.750,-179.771,8.291,149.525
C03196=1127.442,119.956,-57.731,-179.773,8.288,149.525
C03197=1127.447,119.706,-57.711,-179.775,8.284,149.524
C03198=1127.451,119.457,-57.691,-179.777,8.280,149.524
C03199=1127.456,119.208,-57.671,-179.779,8.277,149.524
C03200=1127.461,118.959,-57.652,-179.780,8.274,149.524
C03201=1127.466,118.710,-57.632,-179.782,8.271,149.524
C03202=1127.471,118.460,-57.612,-179.784,8.267,149.523
C03203=1127.475,118.211,-57.592,-179.786,8.263,149.523
C03204=1127.480,117.962,-57.572,-179.788,8.260,149.523
C03205=1127.485,117.713,-57.553,-179.789,8.257,149.522
C03206=1127.489,117.498,-57.536,-179.791,8.254,149.522
C03207=1127.494,117.283,-57.519,-179.793,8.251,149.522
C03208=1127.498,117.068,-57.502,-179.794,8.248,149.522
C03209=1127.502,116.854,-57.484,-179.796,8.245,149.522
C03210=1127.506,116.639,-57.467,-179.798,8.242,149.521
C03211=1127.510,116.425,-57.451,-179.799,8.239,149.521
C03212=1127.514,116.210,-57.434,-179.801,8.236,149.521
C03213=1127.518,115.996,-57.417,-179.803,8.233,149.521
C03214=1127.523,115.746,-57.398,-179.805,8.230,149.520
C03215=1127.528,115.496,-57.378,-179.806,8.226,149.520
C03216=1127.532,115.248,-57.358,-179.809,8.222,149.520
C03217=1127.537,114.999,-57.338,-179.811,8.219,149.520
C03218=1127.542,114.749,-57.319,-179.813,8.215,149.519
C03219=1127.547,114.500,-57.300,-179.814,8.213,149.519
C03220=1127.551,114.251,-57.280,-179.816,8.209,149.519
C03221=1127.556,114.001,-57.261,-179.818,8.205,149.519
C03222=1127.561,113.753,-57.241,-179.820,8.202,149.518
C03223=1127.566,113.504,-57.221,-179.822,8.198,149.518
C03224=1127.571,113.254,-57.201,-179.823,8.194,149.518
C03225=1127.576,113.005,-57.182,-179.826,8.191,149.517
C03226=1127.580,112.756,-57.163,-179.828,8.187,149.517
C03227=1127.585,112.506,-57.143,-179.830,8.184,149.517
C03228=1127.590,112.257,-57.124,-179.832,8.180,149.517
C03229=1127.595,112.008,-57.105,-179.833,8.176,149.516
C03230=1127.600,111.759,-57.086,-179.835,8.173,149.516
C03231=1127.604,111.510,-57.066,-179.837,8.169,149.516
C03232=1127.610,111.261,-57.047,-179.840,8.166,149.516
C03233=1127.614,111.011,-57.027,-179.842,8.162,149.515
C03234=1127.618,110.762,-57.008,-179.843,8.158,149.515
C03235=1127.624,110.513,-56.989,-179.846,8.155,149.515
C03236=1127.628,110.264,-56.969,-179.848,8.151,149.515
C03237=1127.634,110.015,-56.950,-179.851,8.147,149.515
C03238=1127.638,109.765,-56.931,-179.853,8.143,149.514
C03239=1127.643,109.516,-56.912,-179.856,8.139,149.514
C03240=1127.648,109.266,-56.893,-179.859,8.135,149.514
C03241=1127.653,109.018,-56.874,-179.861,8.131,149.514
C03242=1127.658,108.768,-56.854,-179.863,8.127,149.513
C03243=1127.662,108.519,-56.835,-179.865,8.123,149.513
C03244=1127.667,108.270,-56.816,-179.868,8.119,149.513
C03245=1127.672,108.021,-56.796,-179.870,8.116,149.513
C03246=1127.677,107.771,-56.778,-179.873,8.111,149.513
C03247=1127.681,107.522,-56.759,-179.875,8.107,149.512
C03248=1127.687,107.273,-56.739,-179.878,8.104,149.512
C03249=1127.691,107.024,-56.720,-179.880,8.099,149.512
C03250=1127.696,106.774,-56.702,-179.882,8.096,149.512
C03251=1127.700,106.525,-56.683,-179.885,8.092,149.512
C03252=1127.706,106.276,-56.663,-179.887,8.088,149.511
C03253=1127.710,106.028,-56.645,-179.889,8.083,149.511
C03254=1127.715,105.777,-56.626,-179.891,8.080,149.511
C03255=1127.720,105.529,-56.607,-179.894,8.076,149.510
C03256=1127.725,105.279,-56.587,-179.896,8.072,149.510
C03257=1127.730,105.030,-56.569,-179.899,8.068,149.510
C03258=1127.734,104.781,-56.550,-179.900,8.064,149.510
C03259=1127.739,104.532,-56.531,-179.903,8.060,149.509
C03260=1127.745,104.282,-56.512,-179.905,8.056,149.509
C03261=1127.749,104.033,-56.493,-179.907,8.052,149.509
C03262=1127.753,103.818,-56.477,-179.909,8.049,149.508
C03263=1127.757,103.603,-56.461,-179.911,8.045,149.508
C03264=1127.762,103.388,-56.445,-179.913,8.042,149.508
C03265=1127.765,103.174,-56.429,-179.915,8.038,149.508
C03266=1127.770,102.958,-56.413,-179.916,8.036,149.508
C03267=1127.773,102.744,-56.396,-179.918,8.032,149.507
C03268=1127.778,102.529,-56.380,-179.920,8.028,149.507
C03269=1127.782,102.315,-56.364,-179.922,8.025,149.507
C03270=1127.787,102.065,-56.345,-179.924,8.021,149.507
C03271=1127.792,101.816,-56.327,-179.926,8.016,149.506
C03272=1127.797,101.567,-56.308,-179.928,8.013,149.506
C03273=1127.801,101.318,-56.289,-179.930,8.009,149.505
C03274=1127.806,101.069,-56.271,-179.933,8.005,149.505
C03275=1127.811,100.819,-56.251,-179.934,8.001,149.505
C03276=1127.816,100.570,-56.233,-179.936,7.997,149.504
C03277=1127.821,100.321,-56.216,-179.939,7.993,149.504
C03278=1127.826,100.072,-56.196,-179.940,7.989,149.504
C03279=1127.831,99.822,-56.178,-179.942,7.985,149.504
C03280=1127.835,99.573,-56.160,-179.944,7.981,149.503
C03281=1127.841,99.324,-56.141,-179.947,7.977,149.503
C03282=1127.845,99.074,-56.122,-179.948,7.973,149.502
C03283=1127.850,98.825,-56.104,-179.950,7.969,149.502
C03284=1127.855,98.576,-56.085,-179.952,7.965,149.502
C03285=1127.860,98.326,-56.067,-179.954,7.961,149.501
C03286=1127.865,98.077,-56.049,-179.956,7.957,149.501
C03287=1127.869,97.828,-56.030,-179.958,7.954,149.501
C03288=1127.875,97.579,-56.011,-179.960,7.949,149.500
C03289=1127.879,97.329,-55.993,-179.962,7.945,149.500
C03290=1127.884,97.080,-55.975,-179.963,7.941,149.499
C03291=1127.889,96.831,-55.956,-179.965,7.938,149.499
C03292=1127.894,96.582,-55.938,-179.967,7.933,149.499
C03293=1127.899,96.332,-55.919,-179.969,7.929,149.498
C03294=1127.904,96.083,-55.901,-179.971,7.925,149.498
C03295=1127.908,95.834,-55.883,-179.972,7.922,149.498
C03296=1127.913,95.585,-55.865,-179.974,7.918,149.497
C03297=1127.918,95.336,-55.847,-179.976,7.914,149.497
C03298=1127.923,95.086,-55.828,-179.978,7.909,149.496
C03299=1127.928,94.836,-55.810,-179.980,7.906,149.496
C03300=1127.933,94.587,-55.792,-179.981,7.902,149.496
C03301=1127.938,94.338,-55.774,-179.983,7.898,149.495
C03302=1127.943,94.089,-55.756,-179.984,7.894,149.495
C03303=1127.947,93.839,-55.738,-179.986,7.890,149.494
C03304=1127.952,93.590,-55.720,-179.988,7.886,149.494
C03305=1127.957,93.341,-55.700,-179.989,7.882,149.493
C03306=1127.962,93.092,-55.682,-179.991,7.878,149.493
C03307=1127.967,92.843,-55.664,-179.992,7.874,149.493
C03308=1127.972,92.593,-55.646,-179.995,7.870,149.492
C03309=1127.976,92.344,-55.628,-179.996,7.866,149.492
C03310=1127.981,92.094,-55.610,-179.998,7.862,149.491
C03311=1127.986,91.845,-55.592,-179.999,7.858,149.491
C03312=1127.991,91.596,-55.574,179.999,7.854,149.490
C03313=1127.996,91.347,-55.556,179.997,7.850,149.490
C03314=1128.001,91.098,-55.538,179.996,7.846,149.490
C03315=1128.006,90.848,-55.521,179.994,7.843,149.489
C03316=1128.010,90.598,-55.503,179.993,7.839,149.489
C03317=1128.015,90.349,-55.485,179.991,7.835,149.488
C03318=1128.019,90.134,-55.469,179.990,7.832,149.488
C03319=1128.024,89.919,-55.453,179.989,7.829,149.487
C03320=1128.028,89.704,-55.438,179.987,7.825,149.487
C03321=1128.033,89.490,-55.422,179.986,7.822,149.487
C03322=1128.037,89.275,-55.407,179.984,7.818,149.486
C03323=1128.041,89.060,-55.392,179.983,7.815,149.486
C03324=1128.045,88.845,-55.376,179.982,7.812,149.486
C03325=1128.049,88.631,-55.361,179.981,7.808,149.485
C03326=1128.054,88.381,-55.344,179.979,7.804,149.485
C03327=1128.059,88.131,-55.325,179.978,7.800,149.484
C03328=1128.064,87.882,-55.307,179.977,7.797,149.484
C03329=1128.068,87.633,-55.289,179.976,7.793,149.483
C03330=1128.073,87.384,-55.271,179.974,7.789,149.483
C03331=1128.079,87.134,-55.254,179.972,7.785,149.482
C03332=1128.083,86.885,-55.236,179.971,7.781,149.482
C03333=1128.088,86.635,-55.218,179.970,7.777,149.481
C03334=1128.093,86.386,-55.200,179.968,7.773,149.481
C03335=1128.099,86.136,-55.183,179.967,7.770,149.480
C03336=1128.103,85.888,-55.165,179.966,7.765,149.480
C03337=1128.108,85.638,-55.148,179.964,7.762,149.479
C03338=1128.113,85.389,-55.130,179.963,7.758,149.479
C03339=1128.118,85.139,-55.112,179.962,7.754,149.478
C03340=1128.123,84.890,-55.094,179.961,7.750,149.478
C03341=1128.128,84.641,-55.076,179.959,7.746,149.477
C03342=1128.133,84.391,-55.059,179.958,7.742,149.477
C03343=1128.137,84.142,-55.042,179.957,7.739,149.476
C03344=1128.142,83.893,-55.024,179.955,7.735,149.476
C03345=1128.147,83.643,-55.006,179.954,7.731,149.475
C03346=1128.152,83.394,-54.988,179.953,7.727,149.475
C03347=1128.157,83.144,-54.971,179.952,7.723,149.474
C03348=1128.161,82.896,-54.954,179.951,7.720,149.474
C03349=1128.166,82.646,-54.936,179.949,7.716,149.473
C03350=1128.172,82.397,-54.919,179.948,7.712,149.473
C03351=1128.176,82.147,-54.901,179.947,7.708,149.472
C03352=1128.182,81.898,-54.883,179.946,7.704,149.472
C03353=1128.186,81.649,-54.866,179.945,7.701,149.471
C03354=1128.191,81.400,-54.848,179.944,7.697,149.471
C03355=1128.197,81.150,-54.831,179.943,7.693,149.470
C03356=1128.201,80.901,-54.813,179.941,7.690,149.470
C03357=1128.206,80.652,-54.796,179.940,7.685,149.469
C03358=1128.211,80.403,-54.778,179.939,7.682,149.469
C03359=1128.216,80.153,-54.761,179.938,7.678,149.468
C03360=1128.220,79.904,-54.744,179.937,7.675,149.468
C03361=1128.225,79.654,-54.726,179.936,7.670,149.467
C03362=1128.230,79.405,-54.709,179.935,7.667,149.466
C03363=1128.236,79.155,-54.691,179.934,7.663,149.466
C03364=1128.240,78.906,-54.675,179.933,7.660,149.465
C03365=1128.245,78.657,-54.657,179.932,7.656,149.465
C03366=1128.251,78.407,-54.640,179.931,7.652,149.464
C03367=1128.255,78.159,-54.622,179.930,7.648,149.464
C03368=1128.260,77.909,-54.605,179.929,7.645,149.463
C03369=1128.265,77.660,-54.587,179.927,7.641,149.463
C03370=1128.270,77.410,-54.570,179.927,7.637,149.462
C03371=1128.275,77.160,-54.553,179.926,7.633,149.461
C03372=1128.280,76.911,-54.535,179.925,7.630,149.461
C03373=1128.284,76.662,-54.518,179.924,7.626,149.460
C03374=1128.289,76.447,-54.504,179.923,7.623,149.460
C03375=1128.293,76.232,-54.489,179.922,7.619,149.459
C03376=1128.298,76.017,-54.474,179.920,7.616,149.459
C03377=1128.302,75.802,-54.459,179.919,7.613,149.459
C03378=1128.306,75.587,-54.445,179.917,7.609,149.458
C03379=1128.310,75.372,-54.430,179.916,7.606,149.458
C03380=1128.314,75.157,-54.415,179.915,7.603,149.458
C03381=1128.319,74.942,-54.400,179.914,7.599,149.457
C03382=1128.323,74.693,-54.383,179.912,7.595,149.457
C03383=1128.328,74.443,-54.365,179.911,7.591,149.456
C03384=1128.334,74.194,-54.348,179.909,7.587,149.456
C03385=1128.338,73.945,-54.332,179.908,7.583,149.455
C03386=1128.343,73.695,-54.314,179.906,7.579,149.455
C03387=1128.348,73.446,-54.297,179.905,7.575,149.454
C03388=1128.353,73.196,-54.280,179.904,7.571,149.454
C03389=1128.358,72.947,-54.264,179.902,7.567,149.453
C03390=1128.363,72.698,-54.246,179.900,7.563,149.453
C03391=1128.367,72.449,-54.229,179.899,7.559,149.452
C03392=1128.373,72.199,-54.212,179.898,7.555,149.452
C03393=1128.378,71.950,-54.195,179.896,7.551,149.451
C03394=1128.383,71.700,-54.178,179.895,7.547,149.451
C03395=1128.387,71.451,-54.161,179.893,7.543,149.450
C03396=1128.393,71.201,-54.144,179.892,7.539,149.450
C03397=1128.398,70.952,-54.128,179.890,7.535,149.449
C03398=1128.402,70.703,-54.111,179.889,7.532,149.449
C03399=1128.407,70.454,-54.093,179.888,7.527,149.448
C03400=1128.412,70.204,-54.076,179.887,7.523,149.448
C03401=1128.417,69.955,-54.060,179.885,7.520,149.448
C03402=1128.422,69.705,-54.043,179.884,7.516,149.447
C03403=1128.427,69.456,-54.026,179.882,7.511,149.446
C03404=1128.432,69.207,-54.009,179.881,7.507,149.446
C03405=1128.437,68.957,-53.993,179.879,7.504,149.446
C03406=1128.442,68.708,-53.975,179.878,7.500,149.445
C03407=1128.446,68.458,-53.959,179.877,7.495,149.445
C03408=1128.452,68.209,-53.942,179.875,7.491,149.444
C03409=1128.457,67.960,-53.925,179.873,7.488,149.444
C03410=1128.461,67.710,-53.908,179.872,7.483,149.443
C03411=1128.467,67.461,-53.892,179.871,7.479,149.443
C03412=1128.471,67.212,-53.875,179.869,7.475,149.442
C03413=1128.476,66.962,-53.858,179.868,7.472,149.442
C03414=1128.482,66.713,-53.841,179.867,7.467,149.441
C03415=1128.486,66.463,-53.825,179.865,7.463,149.441
C03416=1128.491,66.213,-53.809,179.863,7.459,149.440
C03417=1128.497,65.964,-53.792,179.862,7.455,149.440
C03418=1128.501,65.715,-53.775,179.861,7.451,149.439
C03419=1128.506,65.465,-53.759,179.859,7.447,149.439
C03420=1128.511,65.217,-53.742,179.858,7.443,149.438
C03421=1128.516,64.967,-53.725,179.856,7.439,149.438
C03422=1128.521,64.718,-53.709,179.855,7.435,149.437
C03423=1128.526,64.468,-53.693,179.854,7.431,149.437
C03424=1128.530,64.218,-53.676,179.852,7.427,149.436
C03425=1128.536,63.969,-53.659,179.851,7.423,149.436
C03426=1128.541,63.720,-53.642,179.849,7.419,149.435
C03427=1128.546,63.471,-53.626,179.848,7.415,149.435
C03428=1128.551,63.221,-53.610,179.846,7.411,149.434
C03429=1128.556,62.971,-53.593,179.845,7.407,149.434
C03430=1128.560,62.757,-53.579,179.844,7.404,149.433
C03431=1128.565,62.541,-53.565,179.843,7.400,149.433
C03432=1128.568,62.326,-53.550,179.842,7.397,149.432
C03433=1128.573,62.111,-53.536,179.841,7.393,149.432
C03434=1128.577,61.897,-53.522,179.839,7.390,149.431
C03435=1128.582,61.681,-53.508,179.838,7.386,149.431
C03436=1128.585,61.466,-53.494,179.837,7.383,149.431
C03437=1128.590,61.251,-53.480,179.836,7.379,149.430
C03438=1128.595,61.002,-53.463,179.834,7.375,149.430
C03439=1128.600,60.752,-53.448,179.833,7.372,149.429
C03440=1128.605,60.503,-53.431,179.832,7.367,149.429
C03441=1128.609,60.253,-53.414,179.830,7.363,149.428
C03442=1128.615,60.004,-53.399,179.829,7.359,149.428
C03443=1128.619,59.754,-53.382,179.827,7.355,149.427
C03444=1128.624,59.505,-53.366,179.826,7.351,149.427
C03445=1128.630,59.255,-53.349,179.825,7.347,149.426
C03446=1128.635,59.006,-53.333,179.823,7.343,149.426
C03447=1128.640,58.756,-53.317,179.822,7.339,149.425
C03448=1128.645,58.507,-53.300,179.821,7.335,149.425
C03449=1128.649,58.257,-53.285,179.819,7.331,149.424
C03450=1128.655,58.009,-53.268,179.818,7.327,149.424
C03451=1128.659,57.758,-53.252,179.816,7.323,149.423
C03452=1128.664,57.510,-53.236,179.815,7.319,149.423
C03453=1128.670,57.260,-53.220,179.814,7.315,149.422
C03454=1128.674,57.011,-53.204,179.812,7.311,149.422
C03455=1128.680,56.761,-53.188,179.811,7.306,149.421
C03456=1128.684,56.512,-53.171,179.809,7.302,149.421
C03457=1128.690,56.262,-53.156,179.808,7.298,149.420
C03458=1128.694,56.013,-53.139,179.807,7.294,149.420
C03459=1128.699,55.764,-53.124,179.805,7.290,149.419
C03460=1128.704,55.514,-53.107,179.804,7.286,149.418
C03461=1128.709,55.265,-53.091,179.803,7.282,149.418
C03462=1128.714,55.016,-53.075,179.801,7.278,149.418
C03463=1128.719,54.766,-53.059,179.800,7.274,149.417
C03464=1128.724,54.516,-53.044,179.798,7.270,149.417
C03465=1128.729,54.267,-53.027,179.797,7.266,149.416
C03466=1128.734,54.018,-53.011,179.796,7.262,149.415
C03467=1128.740,53.768,-52.996,179.795,7.257,149.415
C03468=1128.744,53.519,-52.979,179.793,7.254,149.414
C03469=1128.750,53.269,-52.963,179.792,7.249,149.414
C03470=1128.754,53.019,-52.947,179.790,7.245,149.413
C03471=1128.759,52.770,-52.931,179.789,7.241,149.413
C03472=1128.765,52.521,-52.916,179.788,7.237,149.412
C03473=1128.769,52.271,-52.900,179.787,7.233,149.412
C03474=1128.774,52.022,-52.884,179.785,7.229,149.411
C03475=1128.779,51.773,-52.868,179.784,7.225,149.411
C03476=1128.784,51.523,-52.852,179.782,7.221,149.410
C03477=1128.790,51.273,-52.837,179.781,7.217,149.410
C03478=1128.795,51.025,-52.820,179.780,7.212,149.409
C03479=1128.799,50.775,-52.805,179.778,7.209,149.409
C03480=1128.804,50.525,-52.790,179.777,7.204,149.408
C03481=1128.809,50.276,-52.774,179.776,7.200,149.408
C03482=1128.814,50.027,-52.757,179.775,7.196,149.407
C03483=1128.819,49.777,-52.742,179.773,7.192,149.406
C03484=1128.825,49.528,-52.726,179.772,7.188,149.406
C03485=1128.829,49.278,-52.710,179.771,7.183,149.405
C03486=1128.834,49.063,-52.697,179.770,7.180,149.405
C03487=1128.838,48.848,-52.683,179.769,7.177,149.404
C03488=1128.842,48.633,-52.670,179.767,7.173,149.404
C03489=1128.846,48.417,-52.657,179.766,7.170,149.403
C03490=1128.851,48.203,-52.643,179.765,7.166,149.403
C03491=1128.855,47.987,-52.630,179.764,7.163,149.402
C03492=1128.860,47.772,-52.616,179.763,7.159,149.402
C03493=1128.864,47.557,-52.602,179.762,7.156,149.402
C03494=1128.868,47.308,-52.587,179.761,7.151,149.401
C03495=1128.874,47.058,-52.571,179.759,7.147,149.400
C03496=1128.879,46.808,-52.555,179.758,7.143,149.400
C03497=1128.884,46.559,-52.540,179.757,7.139,149.399
C03498=1128.889,46.310,-52.525,179.756,7.135,149.399
C03499=1128.894,46.060,-52.509,179.755,7.131,149.398
C03500=1128.899,45.810,-52.493,179.753,7.127,149.398
C03501=1128.903,45.561,-52.478,179.752,7.122,149.397
C03502=1128.909,45.312,-52.463,179.750,7.119,149.397
C03503=1128.914,45.062,-52.447,179.749,7.114,149.396
C03504=1128.918,44.812,-52.432,179.748,7.110,149.395
C03505=1128.924,44.563,-52.416,179.747,7.106,149.395
C03506=1128.929,44.314,-52.401,179.746,7.102,149.394
C03507=1128.934,44.065,-52.386,179.744,7.098,149.394
C03508=1128.939,43.815,-52.370,179.743,7.093,149.393
C03509=1128.944,43.564,-52.355,179.742,7.089,149.393
C03510=1128.949,43.315,-52.340,179.740,7.085,149.392
C03511=1128.954,43.066,-52.324,179.739,7.080,149.391
C03512=1128.959,42.817,-52.309,179.738,7.076,149.391
C03513=1128.964,42.567,-52.294,179.736,7.072,149.390
C03514=1128.969,42.317,-52.278,179.735,7.068,149.390
C03515=1128.974,42.068,-52.263,179.734,7.063,149.389
C03516=1128.979,41.819,-52.247,179.732,7.059,149.389
C03517=1128.984,41.569,-52.233,179.731,7.055,149.388
C03518=1128.989,41.320,-52.217,179.730,7.051,149.387
C03519=1128.995,41.070,-52.202,179.729,7.047,149.387
C03520=1128.999,40.821,-52.187,179.728,7.043,149.386
C03521=1129.004,40.571,-52.171,179.726,7.038,149.386
C03522=1129.009,40.321,-52.156,179.725,7.034,149.385
C03523=1129.015,40.072,-52.141,179.724,7.030,149.385
C03524=1129.019,39.823,-52.126,179.723,7.026,149.384
C03525=1129.025,39.574,-52.110,179.721,7.022,149.384
C03526=1129.030,39.324,-52.096,179.720,7.017,149.383
C03527=1129.035,39.074,-52.080,179.719,7.013,149.382
C03528=1129.040,38.825,-52.065,179.718,7.009,149.382
C03529=1129.045,38.575,-52.051,179.716,7.005,149.381
C03530=1129.050,38.326,-52.036,179.715,7.001,149.381
C03531=1129.055,38.076,-52.020,179.714,6.996,149.380
C03532=1129.060,37.826,-52.005,179.713,6.992,149.379
C03533=1129.065,37.577,-51.990,179.712,6.988,149.379
C03534=1129.070,37.328,-51.975,179.711,6.984,149.378
C03535=1129.075,37.078,-51.960,179.709,6.979,149.378
C03536=1129.080,36.829,-51.945,179.708,6.974,149.377
C03537=1129.085,36.580,-51.930,179.706,6.970,149.376
C03538=1129.090,36.330,-51.915,179.705,6.966,149.376
C03539=1129.095,36.081,-51.900,179.704,6.962,149.375
C03540=1129.101,35.831,-51.885,179.703,6.957,149.375
C03541=1129.105,35.581,-51.870,179.702,6.953,149.374
C03542=1129.110,35.367,-51.857,179.701,6.950,149.373
C03543=1129.114,35.151,-51.844,179.700,6.946,149.373
C03544=1129.119,34.935,-51.832,179.699,6.943,149.372
C03545=1129.123,34.721,-51.819,179.698,6.939,149.372
C03546=1129.127,34.505,-51.806,179.697,6.935,149.371
C03547=1129.131,34.290,-51.793,179.696,6.931,149.371
C03548=1129.136,34.074,-51.781,179.695,6.928,149.370
C03549=1129.140,33.859,-51.767,179.694,6.924,149.370
C03550=1129.145,33.609,-51.753,179.693,6.919,149.369
C03551=1129.150,33.360,-51.738,179.692,6.915,149.369
C03552=1129.156,33.111,-51.723,179.691,6.911,149.368
C03553=1129.161,32.862,-51.708,179.689,6.906,149.367
C03554=1129.166,32.612,-51.694,179.688,6.903,149.367
C03555=1129.170,32.363,-51.679,179.687,6.898,149.366
C03556=1129.176,32.113,-51.664,179.685,6.893,149.366
C03557=1129.181,31.864,-51.649,179.684,6.889,149.365
C03558=1129.186,31.614,-51.635,179.683,6.885,149.364
C03559=1129.191,31.364,-51.620,179.682,6.880,149.364
C03560=1129.196,31.115,-51.605,179.681,6.876,149.363
C03561=1129.201,30.865,-51.591,179.680,6.872,149.362
C03562=1129.206,30.615,-51.577,179.679,6.867,149.362
C03563=1129.211,30.366,-51.561,179.678,6.863,149.361
C03564=1129.216,30.116,-51.547,179.676,6.859,149.361
C03565=1129.221,29.867,-51.532,179.675,6.855,149.360
C03566=1129.226,29.618,-51.517,179.673,6.850,149.359
C03567=1129.231,29.368,-51.503,179.672,6.845,149.359
C03568=1129.237,29.118,-51.488,179.671,6.841,149.358
C03569=1129.242,28.869,-51.474,179.670,6.837,149.357
C03570=1129.247,28.620,-51.459,179.669,6.832,149.357
C03571=1129.252,28.370,-51.445,179.668,6.828,149.356
C03572=1129.257,28.120,-51.431,179.667,6.824,149.355
C03573=1129.261,27.871,-51.416,179.666,6.819,149.355
C03574=1129.267,27.621,-51.401,179.665,6.815,149.354
C03575=1129.272,27.371,-51.387,179.663,6.810,149.353
C03576=1129.277,27.122,-51.372,179.662,6.806,149.353
C03577=1129.282,26.873,-51.358,179.661,6.801,149.352
C03578=1129.287,26.624,-51.343,179.660,6.797,149.352
C03579=1129.292,26.374,-51.329,179.659,6.793,149.351
C03580=1129.297,26.124,-51.315,179.658,6.788,149.350
C03581=1129.302,25.874,-51.301,179.657,6.784,149.350
C03582=1129.308,25.624,-51.286,179.656,6.780,149.349
C03583=1129.313,25.375,-51.272,179.655,6.774,149.348
C03584=1129.318,25.126,-51.258,179.654,6.770,149.347
C03585=1129.323,24.877,-51.243,179.653,6.766,149.347
C03586=1129.328,24.627,-51.228,179.652,6.761,149.346
C03587=1129.333,24.377,-51.214,179.651,6.757,149.345
C03588=1129.338,24.128,-51.200,179.650,6.753,149.345
C03589=1129.343,23.879,-51.186,179.649,6.748,149.344
C03590=1129.348,23.629,-51.172,179.647,6.743,149.344
C03591=1129.353,23.379,-51.157,179.646,6.739,149.343
C03592=1129.358,23.129,-51.143,179.645,6.735,149.342
C03593=1129.364,22.880,-51.129,179.644,6.730,149.341
C03594=1129.369,22.631,-51.115,179.643,6.726,149.341
C03595=1129.374,22.381,-51.101,179.642,6.721,149.340
C03596=1129.379,22.131,-51.086,179.641,6.717,149.339
C03597=1129.384,21.882,-51.072,179.639,6.712,149.339
C03598=1129.392,21.518,-51.052,179.638,6.705,149.338
C03599=1129.398,21.154,-51.031,179.636,6.699,149.337
C03600=1129.406,20.790,-51.010,179.635,6.692,149.336
C03601=1129.413,20.427,-50.990,179.634,6.685,149.335
C03602=1129.418,20.178,-50.976,179.633,6.681,149.334
C03603=1129.424,19.927,-50.962,179.631,6.677,149.333
C03604=1129.429,19.678,-50.948,179.630,6.673,149.333
C03605=1129.434,19.429,-50.934,179.629,6.667,149.332
C03606=1129.439,19.179,-50.920,179.628,6.663,149.331
C03607=1129.444,18.929,-50.905,179.627,6.658,149.331
C03608=1129.450,18.680,-50.892,179.626,6.654,149.330
C03609=1129.455,18.431,-50.877,179.626,6.649,149.329
C03610=1129.459,18.181,-50.864,179.624,6.644,149.328
C03611=1129.465,17.932,-50.850,179.623,6.640,149.328
C03612=1129.470,17.682,-50.836,179.622,6.635,149.327
C03613=1129.475,17.432,-50.822,179.621,6.631,149.326
C03614=1129.480,17.183,-50.808,179.620,6.627,149.326
C03615=1129.485,16.933,-50.794,179.619,6.621,149.325
C03616=1129.490,16.683,-50.781,179.618,6.617,149.324
C03617=1129.495,16.434,-50.767,179.617,6.612,149.323
C03618=1129.500,16.185,-50.753,179.616,6.608,149.323
C03619=1129.505,15.934,-50.739,179.615,6.603,149.322
C03620=1129.511,15.685,-50.725,179.614,6.598,149.321
C03621=1129.515,15.436,-50.711,179.613,6.594,149.321
C03622=1129.520,15.186,-50.698,179.612,6.589,149.320
C03623=1129.526,14.937,-50.684,179.611,6.585,149.319
C03624=1129.531,14.687,-50.670,179.611,6.580,149.318
C03625=1129.536,14.438,-50.657,179.609,6.575,149.318
C03626=1129.541,14.188,-50.643,179.608,6.571,149.317
C03627=1129.546,13.938,-50.628,179.607,6.566,149.316
C03628=1129.552,13.689,-50.615,179.606,6.562,149.315
C03629=1129.556,13.439,-50.602,179.605,6.556,149.314
C03630=1129.562,13.189,-50.588,179.604,6.552,149.314
C03631=1129.567,12.940,-50.574,179.604,6.547,149.313
C03632=1129.572,12.691,-50.560,179.603,6.543,149.312
C03633=1129.577,12.441,-50.547,179.601,6.538,149.312
C03634=1129.582,12.191,-50.533,179.600,6.533,149.311
C03635=1129.588,11.941,-50.520,179.599,6.529,149.310
